	VAR robtarget Openhole_3455 := [[362.32, -32.55, 173.58], [-0.183051, 0.683002, 0.683002, 0.183051], [0,0,0,0], [9E9, 9E9, 9E9, 9E9, 9E9, 9E9]];
	VAR robtarget Openhole_3456 := [[362.32, -31.54, 174.16], [-0.183051, 0.683002, 0.683002, 0.183051], [0,0,0,0], [9E9, 9E9, 9E9, 9E9, 9E9, 9E9]];
	VAR robtarget Openhole_3457 := [[374.32, -31.54, 174.12], [-0.183051, 0.683002, 0.683002, 0.183051], [0,0,0,0], [9E9, 9E9, 9E9, 9E9, 9E9, 9E9]];
	VAR robtarget Openhole_3458 := [[389.32, -31.54, 174.07], [-0.146559, 0.691752, 0.6724, 0.218811], [0,0,0,0], [9E9, 9E9, 9E9, 9E9, 9E9, 9E9]];
	VAR robtarget Openhole_3459 := [[394.33, -31.54, 174.68], [-0.132991, 0.694488, 0.676088, 0.207135], [0,0,0,0], [9E9, 9E9, 9E9, 9E9, 9E9, 9E9]];
	VAR robtarget Openhole_3460 := [[394.83, -31.57, 174.72], [-0.131528, 0.694766, 0.676427, 0.206027], [0,0,0,0], [9E9, 9E9, 9E9, 9E9, 9E9, 9E9]];
	VAR robtarget Openhole_3461 := [[399.78, -32.12, 175.06], [-0.11586, 0.69755, 0.67957, 0.19541], [0,0,0,0], [9E9, 9E9, 9E9, 9E9, 9E9, 9E9]];
	VAR robtarget Openhole_3462 := [[407.69, -33.18, 175.63], [-0.089063, 0.701475, 0.684337, 0.177998], [0,0,0,0], [9E9, 9E9, 9E9, 9E9, 9E9, 9E9]];
	VAR robtarget Openhole_3463 := [[414.62, -33.85, 176.35], [-0.065291, 0.704086, 0.688563, 0.160875], [0,0,0,0], [9E9, 9E9, 9E9, 9E9, 9E9, 9E9]];
	VAR robtarget Openhole_3464 := [[420.07, -34.09, 177.06], [-0.04691, 0.705549, 0.691908, 0.145819], [0,0,0,0], [9E9, 9E9, 9E9, 9E9, 9E9, 9E9]];
	VAR robtarget Openhole_3465 := [[421.06, -34.1, 177.2], [-0.043641, 0.705759, 0.692517, 0.142901], [0,0,0,0], [9E9, 9E9, 9E9, 9E9, 9E9, 9E9]];
	VAR robtarget Openhole_3466 := [[421.55, -34.1, 177.27], [-0.042014, 0.705857, 0.69282, 0.141422], [0,0,0,0], [9E9, 9E9, 9E9, 9E9, 9E9, 9E9]];
	VAR robtarget Openhole_3467 := [[426.98, -33.88, 178.11], [-0.024649, 0.706677, 0.696114, 0.124201], [0,0,0,0], [9E9, 9E9, 9E9, 9E9, 9E9, 9E9]];
	VAR robtarget Openhole_3468 := [[436.34, -33.07, 179.54], [0.004362, 0.707093, 0.701125, 0.091781], [0,0,0,0], [9E9, 9E9, 9E9, 9E9, 9E9, 9E9]];
	VAR robtarget Openhole_3469 := [[438.32, -33.02, 179.82], [0.010929, 0.707022, 0.701966, 0.085107], [0,0,0,0], [9E9, 9E9, 9E9, 9E9, 9E9, 9E9]];
	VAR robtarget Openhole_3470 := [[438.81, -33.02, 179.88], [0.012627, 0.706994, 0.702162, 0.083481], [0,0,0,0], [9E9, 9E9, 9E9, 9E9, 9E9, 9E9]];
	VAR robtarget Openhole_3471 := [[439.31, -33.03, 179.95], [0.014351, 0.706961, 0.70235, 0.081878], [0,0,0,0], [9E9, 9E9, 9E9, 9E9, 9E9, 9E9]];
	VAR robtarget Openhole_3472 := [[442.77, -33.27, 180.4], [0.026976, 0.706592, 0.703516, 0.071171], [0,0,0,0], [9E9, 9E9, 9E9, 9E9, 9E9, 9E9]];
	VAR robtarget Openhole_3473 := [[447.66, -34.06, 181.06], [0.046306, 0.705589, 0.704776, 0.05736], [0,0,0,0], [9E9, 9E9, 9E9, 9E9, 9E9, 9E9]];
	VAR robtarget Openhole_3474 := [[448.16, -34.12, 181.13], [0.048183, 0.705463, 0.704893, 0.055904], [0,0,0,0], [9E9, 9E9, 9E9, 9E9, 9E9, 9E9]];
	VAR robtarget Openhole_3475 := [[448.65, -34.17, 181.2], [0.050018, 0.705336, 0.705011, 0.054399], [0,0,0,0], [9E9, 9E9, 9E9, 9E9, 9E9, 9E9]];
	VAR robtarget Openhole_3476 := [[449.14, -34.2, 181.27], [0.051809, 0.705206, 0.70513, 0.052839], [0,0,0,0], [9E9, 9E9, 9E9, 9E9, 9E9, 9E9]];
	VAR robtarget Openhole_3477 := [[449.64, -34.22, 181.34], [0.053533, 0.705077, 0.70525, 0.051209], [0,0,0,0], [9E9, 9E9, 9E9, 9E9, 9E9, 9E9]];
	VAR robtarget Openhole_3478 := [[450.13, -34.22, 181.42], [0.055212, 0.704948, 0.70537, 0.049531], [0,0,0,0], [9E9, 9E9, 9E9, 9E9, 9E9, 9E9]];
	VAR robtarget Openhole_3479 := [[450.63, -34.2, 181.49], [0.056822, 0.70482, 0.70549, 0.047788], [0,0,0,0], [9E9, 9E9, 9E9, 9E9, 9E9, 9E9]];
	VAR robtarget Openhole_3480 := [[451.12, -34.17, 181.56], [0.058384, 0.704692, 0.705609, 0.046], [0,0,0,0], [9E9, 9E9, 9E9, 9E9, 9E9, 9E9]];
	VAR robtarget Openhole_3481 := [[451.61, -34.11, 181.63], [0.05987, 0.704568, 0.705727, 0.04415], [0,0,0,0], [9E9, 9E9, 9E9, 9E9, 9E9, 9E9]];
	VAR robtarget Openhole_3482 := [[452.1, -34.05, 181.7], [0.061305, 0.704444, 0.705843, 0.042256], [0,0,0,0], [9E9, 9E9, 9E9, 9E9, 9E9, 9E9]];
	VAR robtarget Openhole_3483 := [[452.59, -33.96, 181.77], [0.062679, 0.704323, 0.705956, 0.040321], [0,0,0,0], [9E9, 9E9, 9E9, 9E9, 9E9, 9E9]];
	VAR robtarget Openhole_3484 := [[460.82, -32.06, 182.74], [0.083784, 0.702126, 0.707082, 0.005917], [0,0,0,0], [9E9, 9E9, 9E9, 9E9, 9E9, 9E9]];
	VAR robtarget Openhole_3485 := [[467.69, -30.95, 183.41], [0.102455, 0.699645, 0.706793, -0.021077], [0,0,0,0], [9E9, 9E9, 9E9, 9E9, 9E9, 9E9]];
	VAR robtarget Openhole_3486 := [[476.61, -29.98, 184.18], [0.127132, 0.695584, 0.705054, -0.053839], [0,0,0,0], [9E9, 9E9, 9E9, 9E9, 9E9, 9E9]];
	VAR robtarget Openhole_3487 := [[487.55, -29.21, 185.05], [0.156769, 0.68951, 0.701222, -0.091037], [0,0,0,0], [9E9, 9E9, 9E9, 9E9, 9E9, 9E9]];
	VAR robtarget Openhole_3488 := [[504.36, -28.38, 186.26], [0.198471, 0.678682, 0.692621, -0.142396], [0,0,0,0], [9E9, 9E9, 9E9, 9E9, 9E9, 9E9]];
	VAR robtarget Openhole_3489 := [[509.36, -28.38, 186.71], [0.183051, 0.683002, 0.683002, -0.183051], [0,0,0,0], [9E9, 9E9, 9E9, 9E9, 9E9, 9E9]];
	VAR robtarget Openhole_3490 := [[536.36, -28.38, 186.62], [0.183051, 0.683002, 0.683002, -0.183051], [0,0,0,0], [9E9, 9E9, 9E9, 9E9, 9E9, 9E9]];
	VAR robtarget Openhole_3491 := [[536.36, -27.26, 185.97], [0.183051, 0.683002, 0.683002, -0.183051], [0,0,0,0], [9E9, 9E9, 9E9, 9E9, 9E9, 9E9]];
	VAR robtarget Openhole_3492 := [[509.36, -27.26, 186.06], [0.183051, 0.683002, 0.683002, -0.183051], [0,0,0,0], [9E9, 9E9, 9E9, 9E9, 9E9, 9E9]];
	VAR robtarget Openhole_3493 := [[504.36, -27.26, 185.66], [0.195255, 0.679614, 0.691939, -0.14567], [0,0,0,0], [9E9, 9E9, 9E9, 9E9, 9E9, 9E9]];
	VAR robtarget Openhole_3494 := [[490.44, -27.87, 184.8], [0.160731, 0.688597, 0.699415, -0.104016], [0,0,0,0], [9E9, 9E9, 9E9, 9E9, 9E9, 9E9]];
	VAR robtarget Openhole_3495 := [[476.49, -28.59, 183.8], [0.122302, 0.69645, 0.704725, -0.057993], [0,0,0,0], [9E9, 9E9, 9E9, 9E9, 9E9, 9E9]];
	VAR robtarget Openhole_3496 := [[464.07, -29.6, 182.8], [0.086303, 0.70182, 0.706981, -0.013352], [0,0,0,0], [9E9, 9E9, 9E9, 9E9, 9E9, 9E9]];
	VAR robtarget Openhole_3497 := [[458.64, -30.3, 182.31], [0.070753, 0.703558, 0.707067, 0.007457], [0,0,0,0], [9E9, 9E9, 9E9, 9E9, 9E9, 9E9]];
	VAR robtarget Openhole_3498 := [[453.73, -31.11, 181.81], [0.057022, 0.704804, 0.706595, 0.026907], [0,0,0,0], [9E9, 9E9, 9E9, 9E9, 9E9, 9E9]];
	VAR robtarget Openhole_3499 := [[452.75, -31.23, 181.7], [0.054101, 0.705034, 0.706441, 0.030675], [0,0,0,0], [9E9, 9E9, 9E9, 9E9, 9E9, 9E9]];
	VAR robtarget Openhole_3500 := [[451.76, -31.32, 181.59], [0.051039, 0.705262, 0.706273, 0.034329], [0,0,0,0], [9E9, 9E9, 9E9, 9E9, 9E9, 9E9]];
	VAR robtarget Openhole_3501 := [[450.76, -31.35, 181.47], [0.0478, 0.705489, 0.706094, 0.037827], [0,0,0,0], [9E9, 9E9, 9E9, 9E9, 9E9, 9E9]];
	VAR robtarget Openhole_3502 := [[450.27, -31.35, 181.41], [0.046116, 0.705601, 0.706002, 0.039513], [0,0,0,0], [9E9, 9E9, 9E9, 9E9, 9E9, 9E9]];
	VAR robtarget Openhole_3503 := [[449.77, -31.34, 181.35], [0.044384, 0.705712, 0.705908, 0.041153], [0,0,0,0], [9E9, 9E9, 9E9, 9E9, 9E9, 9E9]];
	VAR robtarget Openhole_3504 := [[449.27, -31.31, 181.29], [0.042623, 0.705821, 0.705813, 0.042761], [0,0,0,0], [9E9, 9E9, 9E9, 9E9, 9E9, 9E9]];
	VAR robtarget Openhole_3505 := [[445.32, -30.96, 180.84], [0.02795, 0.706554, 0.704968, 0.054953], [0,0,0,0], [9E9, 9E9, 9E9, 9E9, 9E9, 9E9]];
	VAR robtarget Openhole_3506 := [[441.35, -30.75, 180.4], [0.01369, 0.706974, 0.703873, 0.067552], [0,0,0,0], [9E9, 9E9, 9E9, 9E9, 9E9, 9E9]];
	VAR robtarget Openhole_3507 := [[440.85, -30.75, 180.34], [0.011992, 0.707005, 0.703712, 0.069206], [0,0,0,0], [9E9, 9E9, 9E9, 9E9, 9E9, 9E9]];
	VAR robtarget Openhole_3508 := [[440.35, -30.75, 180.29], [0.010316, 0.707032, 0.703546, 0.070877], [0,0,0,0], [9E9, 9E9, 9E9, 9E9, 9E9, 9E9]];
	VAR robtarget Openhole_3509 := [[439.36, -30.78, 180.17], [0.007029, 0.707072, 0.703195, 0.074272], [0,0,0,0], [9E9, 9E9, 9E9, 9E9, 9E9, 9E9]];
	VAR robtarget Openhole_3510 := [[438.37, -30.84, 180.05], [0.003839, 0.707096, 0.702821, 0.077739], [0,0,0,0], [9E9, 9E9, 9E9, 9E9, 9E9, 9E9]];
	VAR robtarget Openhole_3511 := [[432.46, -31.52, 179.27], [-0.013978, 0.706969, 0.700109, 0.099234], [0,0,0,0], [9E9, 9E9, 9E9, 9E9, 9E9, 9E9]];
	VAR robtarget Openhole_3512 := [[426.07, -32.27, 178.34], [-0.032943, 0.706339, 0.696528, 0.121857], [0,0,0,0], [9E9, 9E9, 9E9, 9E9, 9E9, 9E9]];
	VAR robtarget Openhole_3513 := [[421.13, -32.53, 177.64], [-0.048461, 0.705444, 0.693564, 0.137728], [0,0,0,0], [9E9, 9E9, 9E9, 9E9, 9E9, 9E9]];
	VAR robtarget Openhole_3514 := [[419.64, -32.54, 177.44], [-0.05328, 0.705097, 0.692661, 0.142198], [0,0,0,0], [9E9, 9E9, 9E9, 9E9, 9E9, 9E9]];
	VAR robtarget Openhole_3515 := [[419.15, -32.54, 177.38], [-0.0549, 0.704972, 0.69236, 0.143659], [0,0,0,0], [9E9, 9E9, 9E9, 9E9, 9E9, 9E9]];
	VAR robtarget Openhole_3516 := [[413.19, -32.29, 176.69], [-0.074754, 0.703144, 0.688744, 0.1601], [0,0,0,0], [9E9, 9E9, 9E9, 9E9, 9E9, 9E9]];
	VAR robtarget Openhole_3517 := [[404.76, -31.51, 175.95], [-0.103082, 0.699553, 0.683609, 0.180772], [0,0,0,0], [9E9, 9E9, 9E9, 9E9, 9E9, 9E9]];
	VAR robtarget Openhole_3518 := [[397.32, -30.78, 175.42], [-0.126904, 0.695626, 0.678917, 0.197666], [0,0,0,0], [9E9, 9E9, 9E9, 9E9, 9E9, 9E9]];
	VAR robtarget Openhole_3519 := [[394.83, -30.66, 175.2], [-0.134181, 0.694259, 0.677213, 0.203426], [0,0,0,0], [9E9, 9E9, 9E9, 9E9, 9E9, 9E9]];
	VAR robtarget Openhole_3520 := [[389.32, -30.66, 174.58], [-0.149079, 0.691213, 0.673193, 0.216357], [0,0,0,0], [9E9, 9E9, 9E9, 9E9, 9E9, 9E9]];
	VAR robtarget Openhole_3521 := [[362.32, -30.66, 174.67], [-0.183051, 0.683002, 0.683002, 0.183051], [0,0,0,0], [9E9, 9E9, 9E9, 9E9, 9E9, 9E9]];
	VAR robtarget Openhole_3522 := [[362.33, -28.99, 175.63], [-0.183051, 0.683002, 0.683002, 0.183051], [0,0,0,0], [9E9, 9E9, 9E9, 9E9, 9E9, 9E9]];
	VAR robtarget Openhole_3523 := [[374.33, -28.99, 175.59], [-0.183051, 0.683002, 0.683002, 0.183051], [0,0,0,0], [9E9, 9E9, 9E9, 9E9, 9E9, 9E9]];
	VAR robtarget Openhole_3524 := [[389.33, -28.99, 175.55], [-0.153845, 0.690168, 0.674671, 0.211706], [0,0,0,0], [9E9, 9E9, 9E9, 9E9, 9E9, 9E9]];
	VAR robtarget Openhole_3525 := [[394.3, -28.99, 176.02], [-0.140535, 0.693001, 0.678257, 0.199918], [0,0,0,0], [9E9, 9E9, 9E9, 9E9, 9E9, 9E9]];
	VAR robtarget Openhole_3526 := [[394.82, -28.97, 176.09], [-0.139179, 0.693274, 0.67865, 0.198582], [0,0,0,0], [9E9, 9E9, 9E9, 9E9, 9E9, 9E9]];
	VAR robtarget Openhole_3527 := [[396.81, -28.94, 176.29], [-0.133756, 0.694341, 0.680085, 0.193609], [0,0,0,0], [9E9, 9E9, 9E9, 9E9, 9E9, 9E9]];
	VAR robtarget Openhole_3528 := [[397.31, -28.94, 176.34], [-0.132364, 0.694608, 0.680436, 0.19237], [0,0,0,0], [9E9, 9E9, 9E9, 9E9, 9E9, 9E9]];
	VAR robtarget Openhole_3529 := [[403.29, -29.19, 176.8], [-0.114504, 0.697774, 0.684397, 0.177765], [0,0,0,0], [9E9, 9E9, 9E9, 9E9, 9E9, 9E9]];
	VAR robtarget Openhole_3530 := [[414.23, -29.87, 177.64], [-0.079127, 0.702666, 0.691092, 0.149638], [0,0,0,0], [9E9, 9E9, 9E9, 9E9, 9E9, 9E9]];
	VAR robtarget Openhole_3531 := [[417.72, -29.94, 177.98], [-0.067846, 0.703844, 0.693168, 0.13971], [0,0,0,0], [9E9, 9E9, 9E9, 9E9, 9E9, 9E9]];
	VAR robtarget Openhole_3532 := [[418.21, -29.94, 178.03], [-0.06626, 0.703995, 0.693464, 0.138231], [0,0,0,0], [9E9, 9E9, 9E9, 9E9, 9E9, 9E9]];
	VAR robtarget Openhole_3533 := [[423.18, -29.75, 178.6], [-0.050752, 0.705283, 0.696384, 0.122678], [0,0,0,0], [9E9, 9E9, 9E9, 9E9, 9E9, 9E9]];
	VAR robtarget Openhole_3534 := [[427.61, -29.25, 179.16], [-0.037763, 0.706098, 0.698926, 0.107249], [0,0,0,0], [9E9, 9E9, 9E9, 9E9, 9E9, 9E9]];
	VAR robtarget Openhole_3535 := [[431.99, -28.38, 179.74], [-0.025976, 0.70663, 0.701298, 0.09045], [0,0,0,0], [9E9, 9E9, 9E9, 9E9, 9E9, 9E9]];
	VAR robtarget Openhole_3536 := [[436.77, -27.04, 180.33], [-0.014315, 0.706962, 0.703594, 0.070396], [0,0,0,0], [9E9, 9E9, 9E9, 9E9, 9E9, 9E9]];
	VAR robtarget Openhole_3537 := [[439.61, -26.14, 180.64], [-0.0077, 0.707065, 0.70473, 0.057931], [0,0,0,0], [9E9, 9E9, 9E9, 9E9, 9E9, 9E9]];
	VAR robtarget Openhole_3538 := [[441.02, -25.65, 180.77], [-0.004587, 0.707092, 0.705225, 0.05155], [0,0,0,0], [9E9, 9E9, 9E9, 9E9, 9E9, 9E9]];
	VAR robtarget Openhole_3539 := [[441.49, -25.47, 180.81], [-0.003609, 0.707098, 0.70538, 0.04939], [0,0,0,0], [9E9, 9E9, 9E9, 9E9, 9E9, 9E9]];
	VAR robtarget Openhole_3540 := [[441.94, -25.27, 180.86], [-0.002738, 0.707101, 0.705531, 0.047182], [0,0,0,0], [9E9, 9E9, 9E9, 9E9, 9E9, 9E9]];
	VAR robtarget Openhole_3541 := [[442.83, -24.81, 180.94], [-0.00127, 0.707106, 0.705819, 0.04266], [0,0,0,0], [9E9, 9E9, 9E9, 9E9, 9E9, 9E9]];
	VAR robtarget Openhole_3542 := [[443.59, -24.26, 181.01], [-0.000556, 0.707107, 0.706072, 0.038232], [0,0,0,0], [9E9, 9E9, 9E9, 9E9, 9E9, 9E9]];
	VAR robtarget Openhole_3543 := [[445.39, -24.26, 181.1], [0.005592, 0.707085, 0.706376, 0.032131], [0,0,0,0], [9E9, 9E9, 9E9, 9E9, 9E9, 9E9]];
	VAR robtarget Openhole_3544 := [[443.96, -22.2, 181.14], [-0.006277, 0.707079, 0.706469, 0.030031], [0,0,0,0], [9E9, 9E9, 9E9, 9E9, 9E9, 9E9]];
	VAR robtarget Openhole_3545 := [[442.15, -22.2, 181.08], [-0.012413, 0.706998, 0.706183, 0.036126], [0,0,0,0], [9E9, 9E9, 9E9, 9E9, 9E9, 9E9]];
	VAR robtarget Openhole_3546 := [[441.31, -22.66, 181.02], [-0.013707, 0.706974, 0.705945, 0.040513], [0,0,0,0], [9E9, 9E9, 9E9, 9E9, 9E9, 9E9]];
	VAR robtarget Openhole_3547 := [[440.05, -23.46, 180.9], [-0.01527, 0.706942, 0.705512, 0.04746], [0,0,0,0], [9E9, 9E9, 9E9, 9E9, 9E9, 9E9]];
	VAR robtarget Openhole_3548 := [[439.62, -23.72, 180.86], [-0.015855, 0.706929, 0.705354, 0.049754], [0,0,0,0], [9E9, 9E9, 9E9, 9E9, 9E9, 9E9]];
	VAR robtarget Openhole_3549 := [[438.31, -24.43, 180.73], [-0.017925, 0.70688, 0.704844, 0.056527], [0,0,0,0], [9E9, 9E9, 9E9, 9E9, 9E9, 9E9]];
	VAR robtarget Openhole_3550 := [[435.13, -25.85, 180.37], [-0.023883, 0.706703, 0.703452, 0.071802], [0,0,0,0], [9E9, 9E9, 9E9, 9E9, 9E9, 9E9]];
	VAR robtarget Openhole_3551 := [[434.67, -26.03, 180.31], [-0.024835, 0.706671, 0.703232, 0.073926], [0,0,0,0], [9E9, 9E9, 9E9, 9E9, 9E9, 9E9]];
	VAR robtarget Openhole_3552 := [[433.73, -26.37, 180.2], [-0.026829, 0.706598, 0.702778, 0.078118], [0,0,0,0], [9E9, 9E9, 9E9, 9E9, 9E9, 9E9]];
	VAR robtarget Openhole_3553 := [[432.32, -26.83, 180.02], [-0.030072, 0.706467, 0.70207, 0.084249], [0,0,0,0], [9E9, 9E9, 9E9, 9E9, 9E9, 9E9]];
	VAR robtarget Openhole_3554 := [[430.4, -27.35, 179.78], [-0.03475, 0.706252, 0.701076, 0.092158], [0,0,0,0], [9E9, 9E9, 9E9, 9E9, 9E9, 9E9]];
	VAR robtarget Openhole_3555 := [[427, -28.06, 179.36], [-0.043712, 0.705754, 0.699221, 0.105306], [0,0,0,0], [9E9, 9E9, 9E9, 9E9, 9E9, 9E9]];
	VAR robtarget Openhole_3556 := [[422.56, -28.57, 178.84], [-0.056642, 0.704835, 0.69672, 0.120752], [0,0,0,0], [9E9, 9E9, 9E9, 9E9, 9E9, 9E9]];
	VAR robtarget Openhole_3557 := [[417.09, -28.75, 178.28], [-0.073676, 0.703258, 0.693553, 0.137783], [0,0,0,0], [9E9, 9E9, 9E9, 9E9, 9E9, 9E9]];
	VAR robtarget Openhole_3558 := [[416.59, -28.75, 178.24], [-0.07526, 0.70309, 0.693261, 0.139247], [0,0,0,0], [9E9, 9E9, 9E9, 9E9, 9E9, 9E9]];
	VAR robtarget Openhole_3559 := [[408.63, -28.45, 177.61], [-0.100918, 0.699868, 0.688515, 0.161083], [0,0,0,0], [9E9, 9E9, 9E9, 9E9, 9E9, 9E9]];
	VAR robtarget Openhole_3560 := [[399.66, -28.03, 177], [-0.128482, 0.695336, 0.682809, 0.183772], [0,0,0,0], [9E9, 9E9, 9E9, 9E9, 9E9, 9E9]];
	VAR robtarget Openhole_3561 := [[398.16, -28.02, 176.87], [-0.132736, 0.694537, 0.681783, 0.187543], [0,0,0,0], [9E9, 9E9, 9E9, 9E9, 9E9, 9E9]];
	VAR robtarget Openhole_3562 := [[397.66, -28.02, 176.83], [-0.134118, 0.694271, 0.681433, 0.188811], [0,0,0,0], [9E9, 9E9, 9E9, 9E9, 9E9, 9E9]];
	VAR robtarget Openhole_3563 := [[395.18, -28.08, 176.58], [-0.140809, 0.692945, 0.679635, 0.195184], [0,0,0,0], [9E9, 9E9, 9E9, 9E9, 9E9, 9E9]];
	VAR robtarget Openhole_3564 := [[394.33, -28.09, 176.5], [-0.143106, 0.692474, 0.679032, 0.197269], [0,0,0,0], [9E9, 9E9, 9E9, 9E9, 9E9, 9E9]];
	VAR robtarget Openhole_3565 := [[389.33, -28.09, 176.07], [-0.156423, 0.689588, 0.675457, 0.209183], [0,0,0,0], [9E9, 9E9, 9E9, 9E9, 9E9, 9E9]];
	VAR robtarget Openhole_3566 := [[362.33, -28.09, 176.15], [-0.183051, 0.683002, 0.683002, 0.183051], [0,0,0,0], [9E9, 9E9, 9E9, 9E9, 9E9, 9E9]];
	VAR robtarget Openhole_3567 := [[362.33, -27.21, 176.66], [-0.183051, 0.683002, 0.683002, 0.183051], [0,0,0,0], [9E9, 9E9, 9E9, 9E9, 9E9, 9E9]];
	VAR robtarget Openhole_3568 := [[374.33, -27.21, 176.62], [-0.183051, 0.683002, 0.683002, 0.183051], [0,0,0,0], [9E9, 9E9, 9E9, 9E9, 9E9, 9E9]];
	VAR robtarget Openhole_3569 := [[389.33, -27.21, 176.58], [-0.158946, 0.689011, 0.676219, 0.206709], [0,0,0,0], [9E9, 9E9, 9E9, 9E9, 9E9, 9E9]];
	VAR robtarget Openhole_3570 := [[394.26, -27.21, 176.97], [-0.1459, 0.691891, 0.679711, 0.194917], [0,0,0,0], [9E9, 9E9, 9E9, 9E9, 9E9, 9E9]];
	VAR robtarget Openhole_3571 := [[399.8, -27.04, 177.48], [-0.13105, 0.694857, 0.683691, 0.180463], [0,0,0,0], [9E9, 9E9, 9E9, 9E9, 9E9, 9E9]];
	VAR robtarget Openhole_3572 := [[400.3, -27.04, 177.52], [-0.129638, 0.695122, 0.68403, 0.179173], [0,0,0,0], [9E9, 9E9, 9E9, 9E9, 9E9, 9E9]];
	VAR robtarget Openhole_3573 := [[416.26, -27.54, 178.59], [-0.080198, 0.702544, 0.693822, 0.136421], [0,0,0,0], [9E9, 9E9, 9E9, 9E9, 9E9, 9E9]];
	VAR robtarget Openhole_3574 := [[416.76, -27.54, 178.63], [-0.078618, 0.702723, 0.694109, 0.134954], [0,0,0,0], [9E9, 9E9, 9E9, 9E9, 9E9, 9E9]];
	VAR robtarget Openhole_3575 := [[417.26, -27.54, 178.67], [-0.077046, 0.702897, 0.694396, 0.133471], [0,0,0,0], [9E9, 9E9, 9E9, 9E9, 9E9, 9E9]];
	VAR robtarget Openhole_3576 := [[422.73, -27.32, 179.18], [-0.060159, 0.704543, 0.697489, 0.116231], [0,0,0,0], [9E9, 9E9, 9E9, 9E9, 9E9, 9E9]];
	VAR robtarget Openhole_3577 := [[426.68, -26.85, 179.6], [-0.048784, 0.705422, 0.699657, 0.102374], [0,0,0,0], [9E9, 9E9, 9E9, 9E9, 9E9, 9E9]];
	VAR robtarget Openhole_3578 := [[430.07, -26.09, 179.99], [-0.040036, 0.705972, 0.701473, 0.08908], [0,0,0,0], [9E9, 9E9, 9E9, 9E9, 9E9, 9E9]];
	VAR robtarget Openhole_3579 := [[432.91, -25.19, 180.33], [-0.033566, 0.70631, 0.702915, 0.07688], [0,0,0,0], [9E9, 9E9, 9E9, 9E9, 9E9, 9E9]];
	VAR robtarget Openhole_3580 := [[433.37, -25.01, 180.38], [-0.03261, 0.706354, 0.703143, 0.07477], [0,0,0,0], [9E9, 9E9, 9E9, 9E9, 9E9, 9E9]];
	VAR robtarget Openhole_3581 := [[433.83, -24.82, 180.44], [-0.0317, 0.706396, 0.703366, 0.072635], [0,0,0,0], [9E9, 9E9, 9E9, 9E9, 9E9, 9E9]];
	VAR robtarget Openhole_3582 := [[434.29, -24.62, 180.49], [-0.03083, 0.706434, 0.703586, 0.070479], [0,0,0,0], [9E9, 9E9, 9E9, 9E9, 9E9, 9E9]];
	VAR robtarget Openhole_3583 := [[435.19, -24.2, 180.6], [-0.029206, 0.706503, 0.70401, 0.06611], [0,0,0,0], [9E9, 9E9, 9E9, 9E9, 9E9, 9E9]];
	VAR robtarget Openhole_3584 := [[436.52, -23.52, 180.75], [-0.027018, 0.70659, 0.704604, 0.059438], [0,0,0,0], [9E9, 9E9, 9E9, 9E9, 9E9, 9E9]];
	VAR robtarget Openhole_3585 := [[438.24, -22.52, 180.93], [-0.024589, 0.706679, 0.705313, 0.050341], [0,0,0,0], [9E9, 9E9, 9E9, 9E9, 9E9, 9E9]];
	VAR robtarget Openhole_3586 := [[440.79, -20.96, 181.14], [-0.021236, 0.706788, 0.706163, 0.036515], [0,0,0,0], [9E9, 9E9, 9E9, 9E9, 9E9, 9E9]];
	VAR robtarget Openhole_3587 := [[441.58, -20.63, 181.18], [-0.01967, 0.706833, 0.706349, 0.032734], [0,0,0,0], [9E9, 9E9, 9E9, 9E9, 9E9, 9E9]];
	VAR robtarget Openhole_3588 := [[443.72, -20.63, 181.21], [-0.0124, 0.706998, 0.706647, 0.025499], [0,0,0,0], [9E9, 9E9, 9E9, 9E9, 9E9, 9E9]];
	VAR robtarget Openhole_3589 := [[443.53, -19.52, 181.27], [-0.016836, 0.706906, 0.706752, 0.022388], [0,0,0,0], [9E9, 9E9, 9E9, 9E9, 9E9, 9E9]];
	VAR robtarget Openhole_3590 := [[441.39, -19.52, 181.26], [-0.024098, 0.706696, 0.706486, 0.029628], [0,0,0,0], [9E9, 9E9, 9E9, 9E9, 9E9, 9E9]];
	VAR robtarget Openhole_3591 := [[440.77, -19.7, 181.25], [-0.025589, 0.706644, 0.706369, 0.032289], [0,0,0,0], [9E9, 9E9, 9E9, 9E9, 9E9, 9E9]];
	VAR robtarget Openhole_3592 := [[440.31, -19.89, 181.23], [-0.026469, 0.706611, 0.706264, 0.034505], [0,0,0,0], [9E9, 9E9, 9E9, 9E9, 9E9, 9E9]];
	VAR robtarget Openhole_3593 := [[439.86, -20.1, 181.2], [-0.027291, 0.70658, 0.706152, 0.03674], [0,0,0,0], [9E9, 9E9, 9E9, 9E9, 9E9, 9E9]];
	VAR robtarget Openhole_3594 := [[439.41, -20.32, 181.18], [-0.028065, 0.70655, 0.706031, 0.038988], [0,0,0,0], [9E9, 9E9, 9E9, 9E9, 9E9, 9E9]];
	VAR robtarget Openhole_3595 := [[438.97, -20.55, 181.15], [-0.028766, 0.706521, 0.705902, 0.041257], [0,0,0,0], [9E9, 9E9, 9E9, 9E9, 9E9, 9E9]];
	VAR robtarget Openhole_3596 := [[438.54, -20.81, 181.12], [-0.029338, 0.706498, 0.705764, 0.043559], [0,0,0,0], [9E9, 9E9, 9E9, 9E9, 9E9, 9E9]];
	VAR robtarget Openhole_3597 := [[436.45, -22.16, 180.91], [-0.031824, 0.70639, 0.704957, 0.055094], [0,0,0,0], [9E9, 9E9, 9E9, 9E9, 9E9, 9E9]];
	VAR robtarget Openhole_3598 := [[436.02, -22.42, 180.87], [-0.032422, 0.706363, 0.704776, 0.057366], [0,0,0,0], [9E9, 9E9, 9E9, 9E9, 9E9, 9E9]];
	VAR robtarget Openhole_3599 := [[435.15, -22.9, 180.77], [-0.033736, 0.706302, 0.704395, 0.061865], [0,0,0,0], [9E9, 9E9, 9E9, 9E9, 9E9, 9E9]];
	VAR robtarget Openhole_3600 := [[434.26, -23.35, 180.67], [-0.035204, 0.70623, 0.703992, 0.066298], [0,0,0,0], [9E9, 9E9, 9E9, 9E9, 9E9, 9E9]];
	VAR robtarget Openhole_3601 := [[433.36, -23.77, 180.57], [-0.036811, 0.706148, 0.703567, 0.070666], [0,0,0,0], [9E9, 9E9, 9E9, 9E9, 9E9, 9E9]];
	VAR robtarget Openhole_3602 := [[432.44, -24.15, 180.47], [-0.0386, 0.706052, 0.703124, 0.074945], [0,0,0,0], [9E9, 9E9, 9E9, 9E9, 9E9, 9E9]];
	VAR robtarget Openhole_3603 := [[431.98, -24.33, 180.42], [-0.039559, 0.705999, 0.702896, 0.077049], [0,0,0,0], [9E9, 9E9, 9E9, 9E9, 9E9, 9E9]];
	VAR robtarget Openhole_3604 := [[431.04, -24.65, 180.31], [-0.041636, 0.70588, 0.702433, 0.081169], [0,0,0,0], [9E9, 9E9, 9E9, 9E9, 9E9, 9E9]];
	VAR robtarget Openhole_3605 := [[428.64, -25.31, 180.05], [-0.047369, 0.705518, 0.701215, 0.091087], [0,0,0,0], [9E9, 9E9, 9E9, 9E9, 9E9, 9E9]];
	VAR robtarget Openhole_3606 := [[426.69, -25.72, 179.84], [-0.05246, 0.705158, 0.700197, 0.098614], [0,0,0,0], [9E9, 9E9, 9E9, 9E9, 9E9, 9E9]];
	VAR robtarget Openhole_3607 := [[422.74, -26.21, 179.46], [-0.063759, 0.704226, 0.698089, 0.11257], [0,0,0,0], [9E9, 9E9, 9E9, 9E9, 9E9, 9E9]];
	VAR robtarget Openhole_3608 := [[417.77, -26.42, 179.06], [-0.079038, 0.702676, 0.695353, 0.128391], [0,0,0,0], [9E9, 9E9, 9E9, 9E9, 9E9, 9E9]];
	VAR robtarget Openhole_3609 := [[416.77, -26.42, 178.98], [-0.082175, 0.702316, 0.694794, 0.13138], [0,0,0,0], [9E9, 9E9, 9E9, 9E9, 9E9, 9E9]];
	VAR robtarget Openhole_3610 := [[416.27, -26.42, 178.95], [-0.083749, 0.70213, 0.694514, 0.132856], [0,0,0,0], [9E9, 9E9, 9E9, 9E9, 9E9, 9E9]];
	VAR robtarget Openhole_3611 := [[401.3, -26.08, 178.04], [-0.129707, 0.695109, 0.685437, 0.173713], [0,0,0,0], [9E9, 9E9, 9E9, 9E9, 9E9, 9E9]];
	VAR robtarget Openhole_3612 := [[400.8, -26.08, 178.01], [-0.131118, 0.694844, 0.685102, 0.175029], [0,0,0,0], [9E9, 9E9, 9E9, 9E9, 9E9, 9E9]];
	VAR robtarget Openhole_3613 := [[395.33, -26.26, 177.54], [-0.14579, 0.691914, 0.681231, 0.189538], [0,0,0,0], [9E9, 9E9, 9E9, 9E9, 9E9, 9E9]];
	VAR robtarget Openhole_3614 := [[394.83, -26.28, 177.49], [-0.147053, 0.691647, 0.680863, 0.190853], [0,0,0,0], [9E9, 9E9, 9E9, 9E9, 9E9, 9E9]];
	VAR robtarget Openhole_3615 := [[394.33, -26.32, 177.44], [-0.148292, 0.691382, 0.680483, 0.192207], [0,0,0,0], [9E9, 9E9, 9E9, 9E9, 9E9, 9E9]];
	VAR robtarget Openhole_3616 := [[394.33, -26.32, 177.44], [-0.148274, 0.691386, 0.680487, 0.192192], [0,0,0,0], [9E9, 9E9, 9E9, 9E9, 9E9, 9E9]];
	VAR robtarget Openhole_3617 := [[389.33, -26.32, 177.09], [-0.161466, 0.688425, 0.67697, 0.204233], [0,0,0,0], [9E9, 9E9, 9E9, 9E9, 9E9, 9E9]];
	VAR robtarget Openhole_3618 := [[362.33, -26.32, 177.17], [-0.183051, 0.683002, 0.683002, 0.183051], [0,0,0,0], [9E9, 9E9, 9E9, 9E9, 9E9, 9E9]];
	VAR robtarget Openhole_3619 := [[362.34, -24.22, 178.39], [-0.183051, 0.683002, 0.683002, 0.183051], [0,0,0,0], [9E9, 9E9, 9E9, 9E9, 9E9, 9E9]];
	VAR robtarget Openhole_3620 := [[389.34, -24.22, 178.3], [-0.167484, 0.686986, 0.678732, 0.1983], [0,0,0,0], [9E9, 9E9, 9E9, 9E9, 9E9, 9E9]];
	VAR robtarget Openhole_3621 := [[394.34, -24.22, 178.55], [-0.154443, 0.690034, 0.682176, 0.186107], [0,0,0,0], [9E9, 9E9, 9E9, 9E9, 9E9, 9E9]];
	VAR robtarget Openhole_3622 := [[395.31, -24.2, 178.61], [-0.151914, 0.690595, 0.68285, 0.183618], [0,0,0,0], [9E9, 9E9, 9E9, 9E9, 9E9, 9E9]];
	VAR robtarget Openhole_3623 := [[401.29, -23.97, 179.01], [-0.136127, 0.69388, 0.68699, 0.167465], [0,0,0,0], [9E9, 9E9, 9E9, 9E9, 9E9, 9E9]];
	VAR robtarget Openhole_3624 := [[403.28, -23.96, 179.11], [-0.130503, 0.69496, 0.688285, 0.162062], [0,0,0,0], [9E9, 9E9, 9E9, 9E9, 9E9, 9E9]];
	VAR robtarget Openhole_3625 := [[403.78, -23.96, 179.14], [-0.129072, 0.695227, 0.688602, 0.160708], [0,0,0,0], [9E9, 9E9, 9E9, 9E9, 9E9, 9E9]];
	VAR robtarget Openhole_3626 := [[416.77, -24.13, 179.7], [-0.08952, 0.701417, 0.696131, 0.124106], [0,0,0,0], [9E9, 9E9, 9E9, 9E9, 9E9, 9E9]];
	VAR robtarget Openhole_3627 := [[417.27, -24.13, 179.73], [-0.087961, 0.701614, 0.696397, 0.122602], [0,0,0,0], [9E9, 9E9, 9E9, 9E9, 9E9, 9E9]];
	VAR robtarget Openhole_3628 := [[422.76, -23.95, 180.04], [-0.071101, 0.703523, 0.699235, 0.105216], [0,0,0,0], [9E9, 9E9, 9E9, 9E9, 9E9, 9E9]];
	VAR robtarget Openhole_3629 := [[426.72, -23.49, 180.33], [-0.059741, 0.704579, 0.701196, 0.091234], [0,0,0,0], [9E9, 9E9, 9E9, 9E9, 9E9, 9E9]];
	VAR robtarget Openhole_3630 := [[427.7, -23.31, 180.41], [-0.057123, 0.704796, 0.701671, 0.08751], [0,0,0,0], [9E9, 9E9, 9E9, 9E9, 9E9, 9E9]];
	VAR robtarget Openhole_3631 := [[428.19, -23.21, 180.45], [-0.055857, 0.704897, 0.701905, 0.085609], [0,0,0,0], [9E9, 9E9, 9E9, 9E9, 9E9, 9E9]];
	VAR robtarget Openhole_3632 := [[430.12, -22.73, 180.62], [-0.051069, 0.70526, 0.702816, 0.077781], [0,0,0,0], [9E9, 9E9, 9E9, 9E9, 9E9, 9E9]];
	VAR robtarget Openhole_3633 := [[430.6, -22.59, 180.66], [-0.049944, 0.705341, 0.703036, 0.075769], [0,0,0,0], [9E9, 9E9, 9E9, 9E9, 9E9, 9E9]];
	VAR robtarget Openhole_3634 := [[432.02, -22.13, 180.78], [-0.046757, 0.705559, 0.703673, 0.069601], [0,0,0,0], [9E9, 9E9, 9E9, 9E9, 9E9, 9E9]];
	VAR robtarget Openhole_3635 := [[432.49, -21.97, 180.82], [-0.045748, 0.705625, 0.703877, 0.067509], [0,0,0,0], [9E9, 9E9, 9E9, 9E9, 9E9, 9E9]];
	VAR robtarget Openhole_3636 := [[433.88, -21.41, 180.95], [-0.04298, 0.705799, 0.704463, 0.061087], [0,0,0,0], [9E9, 9E9, 9E9, 9E9, 9E9, 9E9]];
	VAR robtarget Openhole_3637 := [[434.78, -20.99, 181.03], [-0.041382, 0.705895, 0.704831, 0.056687], [0,0,0,0], [9E9, 9E9, 9E9, 9E9, 9E9, 9E9]];
	VAR robtarget Openhole_3638 := [[435.23, -20.76, 181.07], [-0.040664, 0.705937, 0.705007, 0.054452], [0,0,0,0], [9E9, 9E9, 9E9, 9E9, 9E9, 9E9]];
	VAR robtarget Openhole_3639 := [[436.1, -20.28, 181.14], [-0.039368, 0.70601, 0.705342, 0.049929], [0,0,0,0], [9E9, 9E9, 9E9, 9E9, 9E9, 9E9]];
	VAR robtarget Openhole_3640 := [[436.54, -20.05, 181.18], [-0.038673, 0.706048, 0.705498, 0.047676], [0,0,0,0], [9E9, 9E9, 9E9, 9E9, 9E9, 9E9]];
	VAR robtarget Openhole_3641 := [[436.99, -19.83, 181.21], [-0.037886, 0.706091, 0.705645, 0.045448], [0,0,0,0], [9E9, 9E9, 9E9, 9E9, 9E9, 9E9]];
	VAR robtarget Openhole_3642 := [[437.9, -19.41, 181.26], [-0.036244, 0.706177, 0.705917, 0.041007], [0,0,0,0], [9E9, 9E9, 9E9, 9E9, 9E9, 9E9]];
	VAR robtarget Openhole_3643 := [[438.36, -19.23, 181.28], [-0.035295, 0.706225, 0.70604, 0.038832], [0,0,0,0], [9E9, 9E9, 9E9, 9E9, 9E9, 9E9]];
	VAR robtarget Openhole_3644 := [[438.84, -19.07, 181.3], [-0.034249, 0.706277, 0.706154, 0.036699], [0,0,0,0], [9E9, 9E9, 9E9, 9E9, 9E9, 9E9]];
	VAR robtarget Openhole_3645 := [[439.31, -18.93, 181.31], [-0.033128, 0.70633, 0.70626, 0.034601], [0,0,0,0], [9E9, 9E9, 9E9, 9E9, 9E9, 9E9]];
	VAR robtarget Openhole_3646 := [[440.28, -18.68, 181.33], [-0.030699, 0.70644, 0.706449, 0.030501], [0,0,0,0], [9E9, 9E9, 9E9, 9E9, 9E9, 9E9]];
	VAR robtarget Openhole_3647 := [[440.77, -18.58, 181.34], [-0.029365, 0.706497, 0.706531, 0.028522], [0,0,0,0], [9E9, 9E9, 9E9, 9E9, 9E9, 9E9]];
	VAR robtarget Openhole_3648 := [[441.27, -18.53, 181.34], [-0.027847, 0.706558, 0.706603, 0.026677], [0,0,0,0], [9E9, 9E9, 9E9, 9E9, 9E9, 9E9]];
	VAR robtarget Openhole_3649 := [[441.35, -18.53, 181.34], [-0.027583, 0.706569, 0.706613, 0.026423], [0,0,0,0], [9E9, 9E9, 9E9, 9E9, 9E9, 9E9]];
	VAR robtarget Openhole_3650 := [[443.12, -18.53, 181.33], [-0.021572, 0.706778, 0.706812, 0.020421], [0,0,0,0], [9E9, 9E9, 9E9, 9E9, 9E9, 9E9]];
	VAR robtarget Openhole_3651 := [[443.2, -17.55, 181.39], [-0.024639, 0.706677, 0.706907, 0.016804], [0,0,0,0], [9E9, 9E9, 9E9, 9E9, 9E9, 9E9]];
	VAR robtarget Openhole_3652 := [[441.43, -17.55, 181.41], [-0.030646, 0.706442, 0.706739, 0.022811], [0,0,0,0], [9E9, 9E9, 9E9, 9E9, 9E9, 9E9]];
	VAR robtarget Openhole_3653 := [[441.37, -17.54, 181.42], [-0.030893, 0.706432, 0.706733, 0.022996], [0,0,0,0], [9E9, 9E9, 9E9, 9E9, 9E9, 9E9]];
	VAR robtarget Openhole_3654 := [[440.87, -17.63, 181.42], [-0.03227, 0.70637, 0.706667, 0.024948], [0,0,0,0], [9E9, 9E9, 9E9, 9E9, 9E9, 9E9]];
	VAR robtarget Openhole_3655 := [[436.92, -18.24, 181.4], [-0.043491, 0.705768, 0.705956, 0.04032], [0,0,0,0], [9E9, 9E9, 9E9, 9E9, 9E9, 9E9]];
	VAR robtarget Openhole_3656 := [[436.43, -18.34, 181.39], [-0.044804, 0.705686, 0.705841, 0.042288], [0,0,0,0], [9E9, 9E9, 9E9, 9E9, 9E9, 9E9]];
	VAR robtarget Openhole_3657 := [[435.94, -18.42, 181.38], [-0.046188, 0.705597, 0.705724, 0.044205], [0,0,0,0], [9E9, 9E9, 9E9, 9E9, 9E9, 9E9]];
	VAR robtarget Openhole_3658 := [[434.95, -18.6, 181.36], [-0.048855, 0.705417, 0.705469, 0.048095], [0,0,0,0], [9E9, 9E9, 9E9, 9E9, 9E9, 9E9]];
	VAR robtarget Openhole_3659 := [[434.46, -18.67, 181.35], [-0.050258, 0.705318, 0.705338, 0.049985], [0,0,0,0], [9E9, 9E9, 9E9, 9E9, 9E9, 9E9]];
	VAR robtarget Openhole_3660 := [[433.97, -18.76, 181.34], [-0.051617, 0.70522, 0.705199, 0.051901], [0,0,0,0], [9E9, 9E9, 9E9, 9E9, 9E9, 9E9]];
	VAR robtarget Openhole_3661 := [[430.5, -19.24, 181.26], [-0.061459, 0.704431, 0.704118, 0.064943], [0,0,0,0], [9E9, 9E9, 9E9, 9E9, 9E9, 9E9]];
	VAR robtarget Openhole_3662 := [[429.51, -19.35, 181.24], [-0.064344, 0.704173, 0.703775, 0.068564], [0,0,0,0], [9E9, 9E9, 9E9, 9E9, 9E9, 9E9]];
	VAR robtarget Openhole_3663 := [[429.01, -19.4, 181.23], [-0.065818, 0.704037, 0.7036, 0.07034], [0,0,0,0], [9E9, 9E9, 9E9, 9E9, 9E9, 9E9]];
	VAR robtarget Openhole_3664 := [[424.02, -19.61, 181.16], [-0.081306, 0.702417, 0.701724, 0.087084], [0,0,0,0], [9E9, 9E9, 9E9, 9E9, 9E9, 9E9]];
	VAR robtarget Openhole_3665 := [[422.52, -19.62, 181.15], [-0.086077, 0.701848, 0.701116, 0.091846], [0,0,0,0], [9E9, 9E9, 9E9, 9E9, 9E9, 9E9]];
	VAR robtarget Openhole_3666 := [[422.02, -19.61, 181.15], [-0.087674, 0.70165, 0.70091, 0.09341], [0,0,0,0], [9E9, 9E9, 9E9, 9E9, 9E9, 9E9]];
	VAR robtarget Openhole_3667 := [[407.52, -19.42, 181.14], [-0.132324, 0.694615, 0.693827, 0.136397], [0,0,0,0], [9E9, 9E9, 9E9, 9E9, 9E9, 9E9]];
	VAR robtarget Openhole_3668 := [[407.02, -19.42, 181.14], [-0.133765, 0.694339, 0.693545, 0.137826], [0,0,0,0], [9E9, 9E9, 9E9, 9E9, 9E9, 9E9]];
	VAR robtarget Openhole_3669 := [[398.02, -19.61, 181.01], [-0.158222, 0.689178, 0.688032, 0.163131], [0,0,0,0], [9E9, 9E9, 9E9, 9E9, 9E9, 9E9]];
	VAR robtarget Openhole_3670 := [[394.34, -19.81, 180.89], [-0.167354, 0.687017, 0.685546, 0.173283], [0,0,0,0], [9E9, 9E9, 9E9, 9E9, 9E9, 9E9]];
	VAR robtarget Openhole_3671 := [[362.34, -19.81, 180.93], [-0.183051, 0.683002, 0.683002, 0.183051], [0,0,0,0], [9E9, 9E9, 9E9, 9E9, 9E9, 9E9]];
	VAR robtarget Openhole_3672 := [[362.35, -16.66, 182.75], [-0.183051, 0.683002, 0.683002, 0.183051], [0,0,0,0], [9E9, 9E9, 9E9, 9E9, 9E9, 9E9]];
	VAR robtarget Openhole_3673 := [[389.35, -16.66, 182.67], [-0.189033, 0.681371, 0.684641, 0.176826], [0,0,0,0], [9E9, 9E9, 9E9, 9E9, 9E9, 9E9]];
	VAR robtarget Openhole_3674 := [[394.35, -16.66, 182.55], [-0.17654, 0.684714, 0.687805, 0.164087], [0,0,0,0], [9E9, 9E9, 9E9, 9E9, 9E9, 9E9]];
	VAR robtarget Openhole_3675 := [[395.16, -16.63, 182.55], [-0.174561, 0.685222, 0.688324, 0.161894], [0,0,0,0], [9E9, 9E9, 9E9, 9E9, 9E9, 9E9]];
	VAR robtarget Openhole_3676 := [[403.65, -16.31, 182.49], [-0.152823, 0.690395, 0.693542, 0.137838], [0,0,0,0], [9E9, 9E9, 9E9, 9E9, 9E9, 9E9]];
	VAR robtarget Openhole_3677 := [[410.15, -16.25, 182.35], [-0.134604, 0.694177, 0.697045, 0.118862], [0,0,0,0], [9E9, 9E9, 9E9, 9E9, 9E9, 9E9]];
	VAR robtarget Openhole_3678 := [[410.65, -16.25, 182.34], [-0.133147, 0.694458, 0.697296, 0.117383], [0,0,0,0], [9E9, 9E9, 9E9, 9E9, 9E9, 9E9]];
	VAR robtarget Openhole_3679 := [[425.64, -16.49, 181.88], [-0.086387, 0.70181, 0.703469, 0.071638], [0,0,0,0], [9E9, 9E9, 9E9, 9E9, 9E9, 9E9]];
	VAR robtarget Openhole_3680 := [[437.63, -16.79, 181.55], [-0.046017, 0.705608, 0.706334, 0.033055], [0,0,0,0], [9E9, 9E9, 9E9, 9E9, 9E9, 9E9]];
	VAR robtarget Openhole_3681 := [[438.13, -16.79, 181.54], [-0.04435, 0.705715, 0.706411, 0.031365], [0,0,0,0], [9E9, 9E9, 9E9, 9E9, 9E9, 9E9]];
	VAR robtarget Openhole_3682 := [[438.63, -16.79, 181.53], [-0.042674, 0.705818, 0.706484, 0.029681], [0,0,0,0], [9E9, 9E9, 9E9, 9E9, 9E9, 9E9]];
	VAR robtarget Openhole_3683 := [[440.13, -16.73, 181.51], [-0.037825, 0.706094, 0.706684, 0.024434], [0,0,0,0], [9E9, 9E9, 9E9, 9E9, 9E9, 9E9]];
	VAR robtarget Openhole_3684 := [[440.63, -16.69, 181.5], [-0.036278, 0.706176, 0.706745, 0.022617], [0,0,0,0], [9E9, 9E9, 9E9, 9E9, 9E9, 9E9]];
	VAR robtarget Openhole_3685 := [[441.11, -16.58, 181.5], [-0.035012, 0.706239, 0.706807, 0.020591], [0,0,0,0], [9E9, 9E9, 9E9, 9E9, 9E9, 9E9]];
	VAR robtarget Openhole_3686 := [[441.66, -16.48, 181.49], [-0.033486, 0.706313, 0.706867, 0.018418], [0,0,0,0], [9E9, 9E9, 9E9, 9E9, 9E9, 9E9]];
	VAR robtarget Openhole_3687 := [[443.56, -16.48, 181.44], [-0.027068, 0.706589, 0.707005, 0.011989], [0,0,0,0], [9E9, 9E9, 9E9, 9E9, 9E9, 9E9]];
	VAR robtarget Openhole_3688 := [[443.93, -15.46, 181.49], [-0.029287, 0.7065, 0.70707, 0.007235], [0,0,0,0], [9E9, 9E9, 9E9, 9E9, 9E9, 9E9]];
	VAR robtarget Openhole_3689 := [[442.03, -15.46, 181.55], [-0.035703, 0.706205, 0.706975, 0.01367], [0,0,0,0], [9E9, 9E9, 9E9, 9E9, 9E9, 9E9]];
	VAR robtarget Openhole_3690 := [[441.46, -15.51, 181.57], [-0.037458, 0.706114, 0.706931, 0.015782], [0,0,0,0], [9E9, 9E9, 9E9, 9E9, 9E9, 9E9]];
	VAR robtarget Openhole_3691 := [[440.97, -15.59, 181.58], [-0.038827, 0.70604, 0.706884, 0.017742], [0,0,0,0], [9E9, 9E9, 9E9, 9E9, 9E9, 9E9]];
	VAR robtarget Openhole_3692 := [[439.97, -15.62, 181.61], [-0.042093, 0.705853, 0.706788, 0.021221], [0,0,0,0], [9E9, 9E9, 9E9, 9E9, 9E9, 9E9]];
	VAR robtarget Openhole_3693 := [[439.47, -15.62, 181.63], [-0.043787, 0.70575, 0.706736, 0.022896], [0,0,0,0], [9E9, 9E9, 9E9, 9E9, 9E9, 9E9]];
	VAR robtarget Openhole_3694 := [[438.97, -15.61, 181.64], [-0.045514, 0.70564, 0.706681, 0.024532], [0,0,0,0], [9E9, 9E9, 9E9, 9E9, 9E9, 9E9]];
	VAR robtarget Openhole_3695 := [[438.47, -15.58, 181.66], [-0.047274, 0.705525, 0.706624, 0.02613], [0,0,0,0], [9E9, 9E9, 9E9, 9E9, 9E9, 9E9]];
	VAR robtarget Openhole_3696 := [[437.48, -15.49, 181.71], [-0.050897, 0.705273, 0.706504, 0.02919], [0,0,0,0], [9E9, 9E9, 9E9, 9E9, 9E9, 9E9]];
	VAR robtarget Openhole_3697 := [[431.51, -14.94, 182], [-0.072517, 0.703378, 0.705526, 0.047249], [0,0,0,0], [9E9, 9E9, 9E9, 9E9, 9E9, 9E9]];
	VAR robtarget Openhole_3698 := [[422.53, -14.66, 182.43], [-0.102246, 0.699676, 0.703052, 0.075619], [0,0,0,0], [9E9, 9E9, 9E9, 9E9, 9E9, 9E9]];
	VAR robtarget Openhole_3699 := [[413.54, -14.6, 182.83], [-0.129852, 0.695082, 0.699492, 0.103495], [0,0,0,0], [9E9, 9E9, 9E9, 9E9, 9E9, 9E9]];
	VAR robtarget Openhole_3700 := [[413.04, -14.6, 182.85], [-0.131325, 0.694805, 0.699265, 0.105014], [0,0,0,0], [9E9, 9E9, 9E9, 9E9, 9E9, 9E9]];
	VAR robtarget Openhole_3701 := [[401.55, -14.77, 183.26], [-0.163243, 0.688006, 0.693301, 0.139045], [0,0,0,0], [9E9, 9E9, 9E9, 9E9, 9E9, 9E9]];
	VAR robtarget Openhole_3702 := [[394.35, -15.07, 183.39], [-0.181155, 0.683508, 0.688896, 0.159443], [0,0,0,0], [9E9, 9E9, 9E9, 9E9, 9E9, 9E9]];
	VAR robtarget Openhole_3703 := [[389.35, -15.07, 183.58], [-0.193533, 0.680107, 0.685795, 0.172295], [0,0,0,0], [9E9, 9E9, 9E9, 9E9, 9E9, 9E9]];
	VAR robtarget Openhole_3704 := [[362.35, -15.07, 183.67], [-0.183051, 0.683002, 0.683002, 0.183051], [0,0,0,0], [9E9, 9E9, 9E9, 9E9, 9E9, 9E9]];
	VAR robtarget Openhole_3705 := [[362.35, -14.11, 184.23], [-0.183051, 0.683002, 0.683002, 0.183051], [0,0,0,0], [9E9, 9E9, 9E9, 9E9, 9E9, 9E9]];
	VAR robtarget Openhole_3706 := [[389.35, -14.11, 184.14], [-0.196264, 0.679324, 0.686481, 0.169539], [0,0,0,0], [9E9, 9E9, 9E9, 9E9, 9E9, 9E9]];
	VAR robtarget Openhole_3707 := [[394.35, -14.11, 183.9], [-0.183956, 0.682759, 0.689544, 0.156617], [0,0,0,0], [9E9, 9E9, 9E9, 9E9, 9E9, 9E9]];
	VAR robtarget Openhole_3708 := [[404.57, -13.71, 183.59], [-0.158197, 0.689183, 0.69556, 0.127266], [0,0,0,0], [9E9, 9E9, 9E9, 9E9, 9E9, 9E9]];
	VAR robtarget Openhole_3709 := [[419.55, -13.55, 182.87], [-0.115078, 0.69768, 0.702399, 0.081456], [0,0,0,0], [9E9, 9E9, 9E9, 9E9, 9E9, 9E9]];
	VAR robtarget Openhole_3710 := [[420.05, -13.55, 182.85], [-0.113543, 0.697931, 0.702581, 0.079876], [0,0,0,0], [9E9, 9E9, 9E9, 9E9, 9E9, 9E9]];
	VAR robtarget Openhole_3711 := [[430.53, -13.69, 182.27], [-0.079851, 0.702584, 0.705587, 0.046339], [0,0,0,0], [9E9, 9E9, 9E9, 9E9, 9E9, 9E9]];
	VAR robtarget Openhole_3712 := [[435.51, -14.05, 181.96], [-0.062314, 0.704356, 0.70643, 0.030925], [0,0,0,0], [9E9, 9E9, 9E9, 9E9, 9E9, 9E9]];
	VAR robtarget Openhole_3713 := [[438.48, -14.4, 181.78], [-0.051201, 0.705251, 0.706761, 0.022123], [0,0,0,0], [9E9, 9E9, 9E9, 9E9, 9E9, 9E9]];
	VAR robtarget Openhole_3714 := [[438.98, -14.45, 181.76], [-0.04939, 0.70538, 0.706807, 0.020588], [0,0,0,0], [9E9, 9E9, 9E9, 9E9, 9E9, 9E9]];
	VAR robtarget Openhole_3715 := [[439.48, -14.47, 181.73], [-0.047627, 0.705501, 0.706852, 0.018992], [0,0,0,0], [9E9, 9E9, 9E9, 9E9, 9E9, 9E9]];
	VAR robtarget Openhole_3716 := [[439.98, -14.49, 181.71], [-0.045913, 0.705615, 0.706894, 0.01734], [0,0,0,0], [9E9, 9E9, 9E9, 9E9, 9E9, 9E9]];
	VAR robtarget Openhole_3717 := [[440.98, -14.49, 181.67], [-0.042535, 0.705826, 0.706969, 0.013974], [0,0,0,0], [9E9, 9E9, 9E9, 9E9, 9E9, 9E9]];
	VAR robtarget Openhole_3718 := [[441.98, -14.53, 181.62], [-0.039029, 0.706029, 0.707025, 0.010732], [0,0,0,0], [9E9, 9E9, 9E9, 9E9, 9E9, 9E9]];
	VAR robtarget Openhole_3719 := [[442.51, -14.54, 181.6], [-0.037183, 0.706128, 0.70705, 0.008962], [0,0,0,0], [9E9, 9E9, 9E9, 9E9, 9E9, 9E9]];
	VAR robtarget Openhole_3720 := [[444.28, -14.54, 181.52], [-0.031181, 0.706419, 0.707101, 0.002936], [0,0,0,0], [9E9, 9E9, 9E9, 9E9, 9E9, 9E9]];
	VAR robtarget Openhole_3721 := [[445.21, -13.31, 181.53], [-0.032234, 0.706372, 0.707093, -0.004392], [0,0,0,0], [9E9, 9E9, 9E9, 9E9, 9E9, 9E9]];
	VAR robtarget Openhole_3722 := [[443.43, -13.31, 181.63], [-0.03824, 0.706072, 0.707105, 0.001641], [0,0,0,0], [9E9, 9E9, 9E9, 9E9, 9E9, 9E9]];
	VAR robtarget Openhole_3723 := [[442.74, -13.1, 181.68], [-0.041273, 0.705901, 0.707099, 0.003287], [0,0,0,0], [9E9, 9E9, 9E9, 9E9, 9E9, 9E9]];
	VAR robtarget Openhole_3724 := [[440.25, -13.05, 181.83], [-0.049868, 0.705346, 0.707012, 0.011561], [0,0,0,0], [9E9, 9E9, 9E9, 9E9, 9E9, 9E9]];
	VAR robtarget Openhole_3725 := [[433.78, -12.57, 182.27], [-0.072956, 0.703333, 0.706392, 0.031776], [0,0,0,0], [9E9, 9E9, 9E9, 9E9, 9E9, 9E9]];
	VAR robtarget Openhole_3726 := [[427.8, -12.45, 182.66], [-0.092777, 0.700994, 0.705246, 0.051262], [0,0,0,0], [9E9, 9E9, 9E9, 9E9, 9E9, 9E9]];
	VAR robtarget Openhole_3727 := [[427.3, -12.45, 182.7], [-0.094372, 0.700781, 0.705125, 0.052902], [0,0,0,0], [9E9, 9E9, 9E9, 9E9, 9E9, 9E9]];
	VAR robtarget Openhole_3728 := [[408.83, -12.69, 183.77], [-0.14945, 0.691133, 0.698238, 0.111639], [0,0,0,0], [9E9, 9E9, 9E9, 9E9, 9E9, 9E9]];
	VAR robtarget Openhole_3729 := [[397.35, -13.06, 184.29], [-0.17938, 0.683976, 0.691975, 0.145503], [0,0,0,0], [9E9, 9E9, 9E9, 9E9, 9E9, 9E9]];
	VAR robtarget Openhole_3730 := [[394.33, -13.23, 184.37], [-0.186569, 0.68205, 0.690114, 0.154087], [0,0,0,0], [9E9, 9E9, 9E9, 9E9, 9E9, 9E9]];
	VAR robtarget Openhole_3731 := [[389.36, -13.23, 184.65], [-0.198759, 0.678598, 0.6871, 0.167014], [0,0,0,0], [9E9, 9E9, 9E9, 9E9, 9E9, 9E9]];
	VAR robtarget Openhole_3732 := [[362.36, -13.23, 184.74], [-0.183051, 0.683002, 0.683002, 0.183051], [0,0,0,0], [9E9, 9E9, 9E9, 9E9, 9E9, 9E9]];
	VAR robtarget Openhole_3733 := [[362.36, -12.34, 185.25], [-0.183051, 0.683002, 0.683002, 0.183051], [0,0,0,0], [9E9, 9E9, 9E9, 9E9, 9E9, 9E9]];
	VAR robtarget Openhole_3734 := [[374.36, -12.34, 185.21], [-0.183051, 0.683002, 0.683002, 0.183051], [0,0,0,0], [9E9, 9E9, 9E9, 9E9, 9E9, 9E9]];
	VAR robtarget Openhole_3735 := [[389.36, -12.34, 185.16], [-0.201251, 0.677863, 0.687709, 0.164489], [0,0,0,0], [9E9, 9E9, 9E9, 9E9, 9E9, 9E9]];
	VAR robtarget Openhole_3736 := [[394.34, -12.34, 184.84], [-0.189119, 0.681347, 0.690688, 0.151493], [0,0,0,0], [9E9, 9E9, 9E9, 9E9, 9E9, 9E9]];
	VAR robtarget Openhole_3737 := [[404.84, -11.88, 184.36], [-0.163039, 0.688054, 0.696696, 0.120889], [0,0,0,0], [9E9, 9E9, 9E9, 9E9, 9E9, 9E9]];
	VAR robtarget Openhole_3738 := [[429.78, -11.27, 182.76], [-0.090335, 0.701313, 0.705929, 0.040793], [0,0,0,0], [9E9, 9E9, 9E9, 9E9, 9E9, 9E9]];
	VAR robtarget Openhole_3739 := [[431.77, -11.25, 182.62], [-0.083929, 0.702108, 0.706284, 0.034099], [0,0,0,0], [9E9, 9E9, 9E9, 9E9, 9E9, 9E9]];
	VAR robtarget Openhole_3740 := [[432.27, -11.25, 182.58], [-0.082304, 0.702301, 0.706363, 0.032434], [0,0,0,0], [9E9, 9E9, 9E9, 9E9, 9E9, 9E9]];
	VAR robtarget Openhole_3741 := [[441.74, -11.43, 181.86], [-0.050325, 0.705314, 0.707106, 0.00103], [0,0,0,0], [9E9, 9E9, 9E9, 9E9, 9E9, 9E9]];
	VAR robtarget Openhole_3742 := [[442.24, -11.45, 181.82], [-0.048561, 0.705437, 0.707107, -0.000574], [0,0,0,0], [9E9, 9E9, 9E9, 9E9, 9E9, 9E9]];
	VAR robtarget Openhole_3743 := [[443.23, -11.52, 181.74], [-0.044965, 0.705676, 0.707097, -0.003712], [0,0,0,0], [9E9, 9E9, 9E9, 9E9, 9E9, 9E9]];
	VAR robtarget Openhole_3744 := [[444.22, -11.62, 181.67], [-0.04128, 0.705901, 0.707075, -0.006756], [0,0,0,0], [9E9, 9E9, 9E9, 9E9, 9E9, 9E9]];
	VAR robtarget Openhole_3745 := [[444.72, -11.69, 181.63], [-0.039394, 0.706009, 0.707059, -0.008227], [0,0,0,0], [9E9, 9E9, 9E9, 9E9, 9E9, 9E9]];
	VAR robtarget Openhole_3746 := [[445.25, -11.83, 181.59], [-0.037109, 0.706132, 0.707042, -0.009568], [0,0,0,0], [9E9, 9E9, 9E9, 9E9, 9E9, 9E9]];
	VAR robtarget Openhole_3747 := [[454.82, -12.87, 180.98], [-0.001006, 0.707106, 0.706056, -0.038538], [0,0,0,0], [9E9, 9E9, 9E9, 9E9, 9E9, 9E9]];
	VAR robtarget Openhole_3748 := [[455.36, -12.53, 180.93], [-0.00035, 0.707107, 0.705889, -0.041479], [0,0,0,0], [9E9, 9E9, 9E9, 9E9, 9E9, 9E9]];
	VAR robtarget Openhole_3749 := [[455.8, -12.3, 180.88], [0.000389, 0.707107, 0.705753, -0.043742], [0,0,0,0], [9E9, 9E9, 9E9, 9E9, 9E9, 9E9]];
	VAR robtarget Openhole_3750 := [[456.25, -12.09, 180.84], [0.001203, 0.707106, 0.70561, -0.045977], [0,0,0,0], [9E9, 9E9, 9E9, 9E9, 9E9, 9E9]];
	VAR robtarget Openhole_3751 := [[456.7, -11.89, 180.8], [0.002055, 0.707104, 0.705462, -0.048195], [0,0,0,0], [9E9, 9E9, 9E9, 9E9, 9E9, 9E9]];
	VAR robtarget Openhole_3752 := [[457.17, -11.7, 180.75], [0.003016, 0.7071, 0.705311, -0.050366], [0,0,0,0], [9E9, 9E9, 9E9, 9E9, 9E9, 9E9]];
	VAR robtarget Openhole_3753 := [[458.11, -11.38, 180.66], [0.005109, 0.707088, 0.704994, -0.054621], [0,0,0,0], [9E9, 9E9, 9E9, 9E9, 9E9, 9E9]];
	VAR robtarget Openhole_3754 := [[464.29, -9.52, 179.93], [0.01985, 0.706828, 0.702416, -0.081314], [0,0,0,0], [9E9, 9E9, 9E9, 9E9, 9E9, 9E9]];
	VAR robtarget Openhole_3755 := [[464.77, -9.39, 179.87], [0.021022, 0.706794, 0.702181, -0.083314], [0,0,0,0], [9E9, 9E9, 9E9, 9E9, 9E9, 9E9]];
	VAR robtarget Openhole_3756 := [[469.61, -8.3, 179.21], [0.033606, 0.706308, 0.699638, -0.102502], [0,0,0,0], [9E9, 9E9, 9E9, 9E9, 9E9, 9E9]];
	VAR robtarget Openhole_3757 := [[474.02, -7.68, 178.61], [0.046177, 0.705597, 0.697122, -0.118413], [0,0,0,0], [9E9, 9E9, 9E9, 9E9, 9E9, 9E9]];
	VAR robtarget Openhole_3758 := [[478.47, -7.38, 178.04], [0.059751, 0.704578, 0.694492, -0.132968], [0,0,0,0], [9E9, 9E9, 9E9, 9E9, 9E9, 9E9]];
	VAR robtarget Openhole_3759 := [[480.96, -7.35, 177.75], [0.067631, 0.703865, 0.693011, -0.140482], [0,0,0,0], [9E9, 9E9, 9E9, 9E9, 9E9, 9E9]];
	VAR robtarget Openhole_3760 := [[481.45, -7.35, 177.69], [0.06922, 0.703711, 0.692713, -0.141946], [0,0,0,0], [9E9, 9E9, 9E9, 9E9, 9E9, 9E9]];
	VAR robtarget Openhole_3761 := [[487.92, -7.59, 177.06], [0.090206, 0.701329, 0.688808, -0.159822], [0,0,0,0], [9E9, 9E9, 9E9, 9E9, 9E9, 9E9]];
	VAR robtarget Openhole_3762 := [[499.86, -8.3, 176.09], [0.127581, 0.695502, 0.681203, -0.189637], [0,0,0,0], [9E9, 9E9, 9E9, 9E9, 9E9, 9E9]];
	VAR robtarget Openhole_3763 := [[501.35, -8.33, 175.94], [0.13184, 0.694707, 0.680164, -0.193332], [0,0,0,0], [9E9, 9E9, 9E9, 9E9, 9E9, 9E9]];
	VAR robtarget Openhole_3764 := [[501.85, -8.33, 175.89], [0.133222, 0.694444, 0.679809, -0.194576], [0,0,0,0], [9E9, 9E9, 9E9, 9E9, 9E9, 9E9]];
	VAR robtarget Openhole_3765 := [[503.83, -8.3, 175.68], [0.138627, 0.693385, 0.678364, -0.199556], [0,0,0,0], [9E9, 9E9, 9E9, 9E9, 9E9, 9E9]];
	VAR robtarget Openhole_3766 := [[504.35, -8.28, 175.61], [0.139966, 0.693116, 0.677966, -0.200903], [0,0,0,0], [9E9, 9E9, 9E9, 9E9, 9E9, 9E9]];
	VAR robtarget Openhole_3767 := [[509.33, -8.28, 175.09], [0.183051, 0.683002, 0.683002, -0.183051], [0,0,0,0], [9E9, 9E9, 9E9, 9E9, 9E9, 9E9]];
	VAR robtarget Openhole_3768 := [[536.33, -8.27, 175.01], [0.183051, 0.683002, 0.683002, -0.183051], [0,0,0,0], [9E9, 9E9, 9E9, 9E9, 9E9, 9E9]];
	VAR robtarget Openhole_3769 := [[536.33, -9.15, 175.51], [0.183051, 0.683002, 0.683002, -0.183051], [0,0,0,0], [9E9, 9E9, 9E9, 9E9, 9E9, 9E9]];
	VAR robtarget Openhole_3770 := [[509.33, -9.15, 175.6], [0.183051, 0.683002, 0.683002, -0.183051], [0,0,0,0], [9E9, 9E9, 9E9, 9E9, 9E9, 9E9]];
	VAR robtarget Openhole_3771 := [[504.33, -9.15, 176.07], [0.142442, 0.692611, 0.678716, -0.198353], [0,0,0,0], [9E9, 9E9, 9E9, 9E9, 9E9, 9E9]];
	VAR robtarget Openhole_3772 := [[503.69, -9.17, 176.15], [0.140778, 0.692951, 0.679197, -0.196703], [0,0,0,0], [9E9, 9E9, 9E9, 9E9, 9E9, 9E9]];
	VAR robtarget Openhole_3773 := [[503.19, -9.2, 176.21], [0.139523, 0.693205, 0.679576, -0.195388], [0,0,0,0], [9E9, 9E9, 9E9, 9E9, 9E9, 9E9]];
	VAR robtarget Openhole_3774 := [[500.21, -9.26, 176.52], [0.131436, 0.694784, 0.681729, -0.187738], [0,0,0,0], [9E9, 9E9, 9E9, 9E9, 9E9, 9E9]];
	VAR robtarget Openhole_3775 := [[499.71, -9.26, 176.56], [0.130032, 0.695048, 0.682076, -0.186474], [0,0,0,0], [9E9, 9E9, 9E9, 9E9, 9E9, 9E9]];
	VAR robtarget Openhole_3776 := [[491.74, -8.94, 177.18], [0.10599, 0.699118, 0.68727, -0.166313], [0,0,0,0], [9E9, 9E9, 9E9, 9E9, 9E9, 9E9]];
	VAR robtarget Openhole_3777 := [[482.78, -8.57, 177.93], [0.077316, 0.702867, 0.692694, -0.142038], [0,0,0,0], [9E9, 9E9, 9E9, 9E9, 9E9, 9E9]];
	VAR robtarget Openhole_3778 := [[481.79, -8.56, 178.03], [0.074151, 0.703208, 0.693285, -0.139127], [0,0,0,0], [9E9, 9E9, 9E9, 9E9, 9E9, 9E9]];
	VAR robtarget Openhole_3779 := [[481.29, -8.56, 178.08], [0.072577, 0.703372, 0.693579, -0.137651], [0,0,0,0], [9E9, 9E9, 9E9, 9E9, 9E9, 9E9]];
	VAR robtarget Openhole_3780 := [[476.32, -8.73, 178.63], [0.057153, 0.704793, 0.69648, -0.122127], [0,0,0,0], [9E9, 9E9, 9E9, 9E9, 9E9, 9E9]];
	VAR robtarget Openhole_3781 := [[471.89, -9.23, 179.18], [0.044252, 0.705721, 0.699011, -0.106695], [0,0,0,0], [9E9, 9E9, 9E9, 9E9, 9E9, 9E9]];
	VAR robtarget Openhole_3782 := [[468.97, -9.8, 179.56], [0.036434, 0.706167, 0.700621, -0.095551], [0,0,0,0], [9E9, 9E9, 9E9, 9E9, 9E9, 9E9]];
	VAR robtarget Openhole_3783 := [[466.57, -10.43, 179.88], [0.030503, 0.706449, 0.701889, -0.08574], [0,0,0,0], [9E9, 9E9, 9E9, 9E9, 9E9, 9E9]];
	VAR robtarget Openhole_3784 := [[463.74, -11.36, 180.24], [0.02415, 0.706694, 0.703289, -0.073382], [0,0,0,0], [9E9, 9E9, 9E9, 9E9, 9E9, 9E9]];
	VAR robtarget Openhole_3785 := [[461.9, -12.1, 180.46], [0.020409, 0.706812, 0.70413, -0.06482], [0,0,0,0], [9E9, 9E9, 9E9, 9E9, 9E9, 9E9]];
	VAR robtarget Openhole_3786 := [[460.54, -12.71, 180.62], [0.01784, 0.706882, 0.704703, -0.058255], [0,0,0,0], [9E9, 9E9, 9E9, 9E9, 9E9, 9E9]];
	VAR robtarget Openhole_3787 := [[459.64, -13.14, 180.72], [0.016278, 0.706919, 0.705057, -0.053804], [0,0,0,0], [9E9, 9E9, 9E9, 9E9, 9E9, 9E9]];
	VAR robtarget Openhole_3788 := [[459.2, -13.37, 180.77], [0.015555, 0.706936, 0.705225, -0.051554], [0,0,0,0], [9E9, 9E9, 9E9, 9E9, 9E9, 9E9]];
	VAR robtarget Openhole_3789 := [[458.76, -13.61, 180.81], [0.014878, 0.70695, 0.705387, -0.049286], [0,0,0,0], [9E9, 9E9, 9E9, 9E9, 9E9, 9E9]];
	VAR robtarget Openhole_3790 := [[457.91, -14.13, 180.9], [0.013724, 0.706974, 0.705693, -0.044687], [0,0,0,0], [9E9, 9E9, 9E9, 9E9, 9E9, 9E9]];
	VAR robtarget Openhole_3791 := [[456.45, -15.03, 181.03], [0.011857, 0.707007, 0.706152, -0.036732], [0,0,0,0], [9E9, 9E9, 9E9, 9E9, 9E9, 9E9]];
	VAR robtarget Openhole_3792 := [[454.01, -15.03, 181.12], [0.00354, 0.707098, 0.706534, -0.028459], [0,0,0,0], [9E9, 9E9, 9E9, 9E9, 9E9, 9E9]];
	VAR robtarget Openhole_3793 := [[454.58, -16.45, 181.17], [0.010306, 0.707032, 0.706644, -0.025565], [0,0,0,0], [9E9, 9E9, 9E9, 9E9, 9E9, 9E9]];
	VAR robtarget Openhole_3794 := [[457.02, -16.45, 181.11], [0.018611, 0.706862, 0.706297, -0.03384], [0,0,0,0], [9E9, 9E9, 9E9, 9E9, 9E9, 9E9]];
	VAR robtarget Openhole_3795 := [[457.6, -16.2, 181.08], [0.019698, 0.706832, 0.706157, -0.03664], [0,0,0,0], [9E9, 9E9, 9E9, 9E9, 9E9, 9E9]];
	VAR robtarget Openhole_3796 := [[458.48, -15.74, 181.01], [0.021141, 0.706791, 0.705907, -0.041176], [0,0,0,0], [9E9, 9E9, 9E9, 9E9, 9E9, 9E9]];
	VAR robtarget Openhole_3797 := [[458.92, -15.49, 180.98], [0.021766, 0.706772, 0.705769, -0.043468], [0,0,0,0], [9E9, 9E9, 9E9, 9E9, 9E9, 9E9]];
	VAR robtarget Openhole_3798 := [[459.34, -15.23, 180.94], [0.022319, 0.706754, 0.705624, -0.045774], [0,0,0,0], [9E9, 9E9, 9E9, 9E9, 9E9, 9E9]];
	VAR robtarget Openhole_3799 := [[460.18, -14.69, 180.85], [0.023321, 0.706722, 0.705308, -0.0504], [0,0,0,0], [9E9, 9E9, 9E9, 9E9, 9E9, 9E9]];
	VAR robtarget Openhole_3800 := [[461.04, -14.18, 180.76], [0.024495, 0.706682, 0.704967, -0.054971], [0,0,0,0], [9E9, 9E9, 9E9, 9E9, 9E9, 9E9]];
	VAR robtarget Openhole_3801 := [[463.23, -13.02, 180.5], [0.027995, 0.706552, 0.704004, -0.066168], [0,0,0,0], [9E9, 9E9, 9E9, 9E9, 9E9, 9E9]];
	VAR robtarget Openhole_3802 := [[463.68, -12.81, 180.44], [0.028797, 0.70652, 0.703795, -0.068361], [0,0,0,0], [9E9, 9E9, 9E9, 9E9, 9E9, 9E9]];
	VAR robtarget Openhole_3803 := [[465.05, -12.22, 180.27], [0.031419, 0.706408, 0.703136, -0.074829], [0,0,0,0], [9E9, 9E9, 9E9, 9E9, 9E9, 9E9]];
	VAR robtarget Openhole_3804 := [[465.51, -12.04, 180.21], [0.032363, 0.706366, 0.702908, -0.076946], [0,0,0,0], [9E9, 9E9, 9E9, 9E9, 9E9, 9E9]];
	VAR robtarget Openhole_3805 := [[468.83, -10.99, 179.79], [0.039929, 0.705979, 0.701205, -0.091165], [0,0,0,0], [9E9, 9E9, 9E9, 9E9, 9E9, 9E9]];
	VAR robtarget Openhole_3806 := [[469.79, -10.75, 179.67], [0.042336, 0.705838, 0.70069, -0.095043], [0,0,0,0], [9E9, 9E9, 9E9, 9E9, 9E9, 9E9]];
	VAR robtarget Openhole_3807 := [[473.7, -10.06, 179.2], [0.052944, 0.705122, 0.698549, -0.109681], [0,0,0,0], [9E9, 9E9, 9E9, 9E9, 9E9, 9E9]];
	VAR robtarget Openhole_3808 := [[478.16, -9.69, 178.71], [0.066189, 0.704002, 0.696034, -0.124644], [0,0,0,0], [9E9, 9E9, 9E9, 9E9, 9E9, 9E9]];
	VAR robtarget Openhole_3809 := [[482.14, -9.61, 178.33], [0.078623, 0.702722, 0.693741, -0.136831], [0,0,0,0], [9E9, 9E9, 9E9, 9E9, 9E9, 9E9]];
	VAR robtarget Openhole_3810 := [[482.64, -9.62, 178.29], [0.080197, 0.702544, 0.693451, -0.138297], [0,0,0,0], [9E9, 9E9, 9E9, 9E9, 9E9, 9E9]];
	VAR robtarget Openhole_3811 := [[494.09, -10.02, 177.42], [0.116232, 0.697488, 0.686503, -0.169449], [0,0,0,0], [9E9, 9E9, 9E9, 9E9, 9E9, 9E9]];
	VAR robtarget Openhole_3812 := [[499.58, -10.13, 177], [0.132245, 0.69463, 0.682862, -0.183576], [0,0,0,0], [9E9, 9E9, 9E9, 9E9, 9E9, 9E9]];
	VAR robtarget Openhole_3813 := [[500.08, -10.12, 176.95], [0.133631, 0.694365, 0.682515, -0.18486], [0,0,0,0], [9E9, 9E9, 9E9, 9E9, 9E9, 9E9]];
	VAR robtarget Openhole_3814 := [[503.56, -10.02, 176.6], [0.142895, 0.692518, 0.679991, -0.193937], [0,0,0,0], [9E9, 9E9, 9E9, 9E9, 9E9, 9E9]];
	VAR robtarget Openhole_3815 := [[504.33, -10, 176.53], [0.144956, 0.692089, 0.679431, -0.195891], [0,0,0,0], [9E9, 9E9, 9E9, 9E9, 9E9, 9E9]];
	VAR robtarget Openhole_3816 := [[509.33, -10, 176.09], [0.183051, 0.683002, 0.683002, -0.183051], [0,0,0,0], [9E9, 9E9, 9E9, 9E9, 9E9, 9E9]];
	VAR robtarget Openhole_3817 := [[536.33, -10, 176.01], [0.183051, 0.683002, 0.683002, -0.183051], [0,0,0,0], [9E9, 9E9, 9E9, 9E9, 9E9, 9E9]];
	VAR robtarget Openhole_3818 := [[536.33, -10.89, 176.52], [0.183051, 0.683002, 0.683002, -0.183051], [0,0,0,0], [9E9, 9E9, 9E9, 9E9, 9E9, 9E9]];
	VAR robtarget Openhole_3819 := [[524.33, -10.89, 176.55], [0.183051, 0.683002, 0.683002, -0.183051], [0,0,0,0], [9E9, 9E9, 9E9, 9E9, 9E9, 9E9]];
	VAR robtarget Openhole_3820 := [[509.33, -10.89, 176.6], [0.183051, 0.683002, 0.683002, -0.183051], [0,0,0,0], [9E9, 9E9, 9E9, 9E9, 9E9, 9E9]];
	VAR robtarget Openhole_3821 := [[504.39, -10.89, 176.99], [0.147705, 0.691508, 0.680116, -0.193501], [0,0,0,0], [9E9, 9E9, 9E9, 9E9, 9E9, 9E9]];
	VAR robtarget Openhole_3822 := [[498.87, -11.14, 177.54], [0.133281, 0.694432, 0.684139, -0.178758], [0,0,0,0], [9E9, 9E9, 9E9, 9E9, 9E9, 9E9]];
	VAR robtarget Openhole_3823 := [[497.37, -11.14, 177.66], [0.129086, 0.695224, 0.685156, -0.174817], [0,0,0,0], [9E9, 9E9, 9E9, 9E9, 9E9, 9E9]];
	VAR robtarget Openhole_3824 := [[496.87, -11.14, 177.69], [0.127662, 0.695487, 0.685489, -0.173507], [0,0,0,0], [9E9, 9E9, 9E9, 9E9, 9E9, 9E9]];
	VAR robtarget Openhole_3825 := [[482.41, -10.79, 178.68], [0.083264, 0.702187, 0.694311, -0.13391], [0,0,0,0], [9E9, 9E9, 9E9, 9E9, 9E9, 9E9]];
	VAR robtarget Openhole_3826 := [[481.91, -10.8, 178.72], [0.081702, 0.702371, 0.694596, -0.132425], [0,0,0,0], [9E9, 9E9, 9E9, 9E9, 9E9, 9E9]];
	VAR robtarget Openhole_3827 := [[476.44, -10.97, 179.2], [0.064808, 0.704131, 0.69765, -0.115261], [0,0,0,0], [9E9, 9E9, 9E9, 9E9, 9E9, 9E9]];
	VAR robtarget Openhole_3828 := [[472.49, -11.44, 179.61], [0.053485, 0.705081, 0.6998, -0.101393], [0,0,0,0], [9E9, 9E9, 9E9, 9E9, 9E9, 9E9]];
	VAR robtarget Openhole_3829 := [[471.02, -11.7, 179.77], [0.049521, 0.705371, 0.700577, -0.095873], [0,0,0,0], [9E9, 9E9, 9E9, 9E9, 9E9, 9E9]];
	VAR robtarget Openhole_3830 := [[470.53, -11.8, 179.83], [0.048255, 0.705458, 0.700833, -0.093985], [0,0,0,0], [9E9, 9E9, 9E9, 9E9, 9E9, 9E9]];
	VAR robtarget Openhole_3831 := [[469.57, -12.03, 179.94], [0.045816, 0.705621, 0.701339, -0.090132], [0,0,0,0], [9E9, 9E9, 9E9, 9E9, 9E9, 9E9]];
	VAR robtarget Openhole_3832 := [[468.61, -12.29, 180.05], [0.043501, 0.705767, 0.701835, -0.086183], [0,0,0,0], [9E9, 9E9, 9E9, 9E9, 9E9, 9E9]];
	VAR robtarget Openhole_3833 := [[467.66, -12.58, 180.16], [0.041312, 0.705899, 0.702319, -0.082142], [0,0,0,0], [9E9, 9E9, 9E9, 9E9, 9E9, 9E9]];
	VAR robtarget Openhole_3834 := [[466.25, -13.07, 180.33], [0.038288, 0.706069, 0.70302, -0.075913], [0,0,0,0], [9E9, 9E9, 9E9, 9E9, 9E9, 9E9]];
	VAR robtarget Openhole_3835 := [[465.79, -13.26, 180.39], [0.037363, 0.706119, 0.703246, -0.073789], [0,0,0,0], [9E9, 9E9, 9E9, 9E9, 9E9, 9E9]];
	VAR robtarget Openhole_3836 := [[465.33, -13.45, 180.44], [0.036484, 0.706165, 0.703468, -0.071641], [0,0,0,0], [9E9, 9E9, 9E9, 9E9, 9E9, 9E9]];
	VAR robtarget Openhole_3837 := [[464.88, -13.66, 180.5], [0.035662, 0.706207, 0.703686, -0.069467], [0,0,0,0], [9E9, 9E9, 9E9, 9E9, 9E9, 9E9]];
	VAR robtarget Openhole_3838 := [[463.11, -14.56, 180.71], [0.032767, 0.706347, 0.704506, -0.060588], [0,0,0,0], [9E9, 9E9, 9E9, 9E9, 9E9, 9E9]];
	VAR robtarget Openhole_3839 := [[461.82, -15.31, 180.86], [0.030959, 0.706429, 0.705059, -0.053777], [0,0,0,0], [9E9, 9E9, 9E9, 9E9, 9E9, 9E9]];
	VAR robtarget Openhole_3840 := [[460.15, -16.4, 181.03], [0.029002, 0.706512, 0.705703, -0.044533], [0,0,0,0], [9E9, 9E9, 9E9, 9E9, 9E9, 9E9]];
	VAR robtarget Openhole_3841 := [[459.72, -16.65, 181.06], [0.028409, 0.706536, 0.705844, -0.042237], [0,0,0,0], [9E9, 9E9, 9E9, 9E9, 9E9, 9E9]];
	VAR robtarget Openhole_3842 := [[459.27, -16.88, 181.1], [0.027653, 0.706566, 0.705975, -0.039985], [0,0,0,0], [9E9, 9E9, 9E9, 9E9, 9E9, 9E9]];
	VAR robtarget Openhole_3843 := [[458.82, -17.08, 181.12], [0.026805, 0.706599, 0.706098, -0.037763], [0,0,0,0], [9E9, 9E9, 9E9, 9E9, 9E9, 9E9]];
	VAR robtarget Openhole_3844 := [[458.35, -17.26, 181.15], [0.02585, 0.706634, 0.706211, -0.035581], [0,0,0,0], [9E9, 9E9, 9E9, 9E9, 9E9, 9E9]];
	VAR robtarget Openhole_3845 := [[457.88, -17.43, 181.17], [0.024838, 0.70667, 0.706316, -0.033423], [0,0,0,0], [9E9, 9E9, 9E9, 9E9, 9E9, 9E9]];
	VAR robtarget Openhole_3846 := [[457.27, -17.6, 181.19], [0.02333, 0.706722, 0.706436, -0.030789], [0,0,0,0], [9E9, 9E9, 9E9, 9E9, 9E9, 9E9]];
	VAR robtarget Openhole_3847 := [[454.82, -17.6, 181.23], [0.015035, 0.706947, 0.706748, -0.022509], [0,0,0,0], [9E9, 9E9, 9E9, 9E9, 9E9, 9E9]];
	VAR robtarget Openhole_3848 := [[454.9, -18.58, 181.28], [0.018612, 0.706862, 0.706839, -0.019447], [0,0,0,0], [9E9, 9E9, 9E9, 9E9, 9E9, 9E9]];
	VAR robtarget Openhole_3849 := [[457.35, -18.58, 181.27], [0.0269, 0.706595, 0.706563, -0.027733], [0,0,0,0], [9E9, 9E9, 9E9, 9E9, 9E9, 9E9]];
	VAR robtarget Openhole_3850 := [[457.46, -18.57, 181.27], [0.027297, 0.70658, 0.706547, -0.028138], [0,0,0,0], [9E9, 9E9, 9E9, 9E9, 9E9, 9E9]];
	VAR robtarget Openhole_3851 := [[457.96, -18.57, 181.26], [0.02897, 0.706513, 0.706477, -0.029843], [0,0,0,0], [9E9, 9E9, 9E9, 9E9, 9E9, 9E9]];
	VAR robtarget Openhole_3852 := [[458.45, -18.46, 181.25], [0.030247, 0.70646, 0.706389, -0.031858], [0,0,0,0], [9E9, 9E9, 9E9, 9E9, 9E9, 9E9]];
	VAR robtarget Openhole_3853 := [[459.42, -18.22, 181.22], [0.03269, 0.706351, 0.706192, -0.035949], [0,0,0,0], [9E9, 9E9, 9E9, 9E9, 9E9, 9E9]];
	VAR robtarget Openhole_3854 := [[460.37, -17.92, 181.18], [0.034892, 0.706245, 0.705965, -0.040162], [0,0,0,0], [9E9, 9E9, 9E9, 9E9, 9E9, 9E9]];
	VAR robtarget Openhole_3855 := [[460.84, -17.74, 181.16], [0.035843, 0.706198, 0.705838, -0.042335], [0,0,0,0], [9E9, 9E9, 9E9, 9E9, 9E9, 9E9]];
	VAR robtarget Openhole_3856 := [[461.3, -17.54, 181.13], [0.036739, 0.706152, 0.705703, -0.044529], [0,0,0,0], [9E9, 9E9, 9E9, 9E9, 9E9, 9E9]];
	VAR robtarget Openhole_3857 := [[462.19, -17.09, 181.06], [0.038176, 0.706076, 0.705405, -0.049032], [0,0,0,0], [9E9, 9E9, 9E9, 9E9, 9E9, 9E9]];
	VAR robtarget Openhole_3858 := [[463.94, -16.14, 180.9], [0.040871, 0.705925, 0.70472, -0.058046], [0,0,0,0], [9E9, 9E9, 9E9, 9E9, 9E9, 9E9]];
	VAR robtarget Openhole_3859 := [[464.83, -15.7, 180.81], [0.04234, 0.705838, 0.70434, -0.06249], [0,0,0,0], [9E9, 9E9, 9E9, 9E9, 9E9, 9E9]];
	VAR robtarget Openhole_3860 := [[465.73, -15.28, 180.71], [0.043936, 0.70574, 0.703938, -0.066871], [0,0,0,0], [9E9, 9E9, 9E9, 9E9, 9E9, 9E9]];
	VAR robtarget Openhole_3861 := [[466.19, -15.08, 180.66], [0.044792, 0.705687, 0.703729, -0.069033], [0,0,0,0], [9E9, 9E9, 9E9, 9E9, 9E9, 9E9]];
	VAR robtarget Openhole_3862 := [[466.65, -14.89, 180.61], [0.045688, 0.705629, 0.703516, -0.071174], [0,0,0,0], [9E9, 9E9, 9E9, 9E9, 9E9, 9E9]];
	VAR robtarget Openhole_3863 := [[467.12, -14.71, 180.56], [0.046638, 0.705567, 0.703299, -0.073287], [0,0,0,0], [9E9, 9E9, 9E9, 9E9, 9E9, 9E9]];
	VAR robtarget Openhole_3864 := [[467.59, -14.54, 180.51], [0.047636, 0.7055, 0.703078, -0.075373], [0,0,0,0], [9E9, 9E9, 9E9, 9E9, 9E9, 9E9]];
	VAR robtarget Openhole_3865 := [[468.53, -14.24, 180.42], [0.049753, 0.705354, 0.702627, -0.079469], [0,0,0,0], [9E9, 9E9, 9E9, 9E9, 9E9, 9E9]];
	VAR robtarget Openhole_3866 := [[469.49, -13.97, 180.32], [0.052017, 0.705191, 0.702163, -0.083468], [0,0,0,0], [9E9, 9E9, 9E9, 9E9, 9E9, 9E9]];
	VAR robtarget Openhole_3867 := [[470.46, -13.73, 180.22], [0.054392, 0.705012, 0.701687, -0.087379], [0,0,0,0], [9E9, 9E9, 9E9, 9E9, 9E9, 9E9]];
	VAR robtarget Openhole_3868 := [[470.94, -13.62, 180.18], [0.055622, 0.704916, 0.701445, -0.089299], [0,0,0,0], [9E9, 9E9, 9E9, 9E9, 9E9, 9E9]];
	VAR robtarget Openhole_3869 := [[471.92, -13.42, 180.08], [0.058168, 0.70471, 0.700955, -0.093069], [0,0,0,0], [9E9, 9E9, 9E9, 9E9, 9E9, 9E9]];
	VAR robtarget Openhole_3870 := [[475.87, -12.91, 179.74], [0.069332, 0.7037, 0.698936, -0.107185], [0,0,0,0], [9E9, 9E9, 9E9, 9E9, 9E9, 9E9]];
	VAR robtarget Openhole_3871 := [[480.85, -12.71, 179.39], [0.084529, 0.702036, 0.696304, -0.12313], [0,0,0,0], [9E9, 9E9, 9E9, 9E9, 9E9, 9E9]];
	VAR robtarget Openhole_3872 := [[482.35, -12.7, 179.29], [0.08918, 0.701461, 0.695487, -0.127663], [0,0,0,0], [9E9, 9E9, 9E9, 9E9, 9E9, 9E9]];
	VAR robtarget Openhole_3873 := [[482.85, -12.7, 179.26], [0.090734, 0.701261, 0.695212, -0.129152], [0,0,0,0], [9E9, 9E9, 9E9, 9E9, 9E9, 9E9]];
	VAR robtarget Openhole_3874 := [[495.33, -12.89, 178.59], [0.128579, 0.695318, 0.687801, -0.164101], [0,0,0,0], [9E9, 9E9, 9E9, 9E9, 9E9, 9E9]];
	VAR robtarget Openhole_3875 := [[495.83, -12.89, 178.56], [0.13, 0.695054, 0.687477, -0.165453], [0,0,0,0], [9E9, 9E9, 9E9, 9E9, 9E9, 9E9]];
	VAR robtarget Openhole_3876 := [[501.81, -12.75, 178.13], [0.146208, 0.691826, 0.683391, -0.181596], [0,0,0,0], [9E9, 9E9, 9E9, 9E9, 9E9, 9E9]];
	VAR robtarget Openhole_3877 := [[504.34, -12.58, 177.89], [0.152514, 0.690463, 0.68153, -0.188461], [0,0,0,0], [9E9, 9E9, 9E9, 9E9, 9E9, 9E9]];
	VAR robtarget Openhole_3878 := [[509.33, -12.58, 177.58], [0.183051, 0.683002, 0.683002, -0.183051], [0,0,0,0], [9E9, 9E9, 9E9, 9E9, 9E9, 9E9]];
	VAR robtarget Openhole_3879 := [[536.33, -12.58, 177.5], [0.183051, 0.683002, 0.683002, -0.183051], [0,0,0,0], [9E9, 9E9, 9E9, 9E9, 9E9, 9E9]];
	VAR robtarget Openhole_3880 := [[536.34, -16.49, 179.75], [0.183051, 0.683002, 0.683002, -0.183051], [0,0,0,0], [9E9, 9E9, 9E9, 9E9, 9E9, 9E9]];
	VAR robtarget Openhole_3881 := [[509.34, -16.49, 179.84], [0.183051, 0.683002, 0.683002, -0.183051], [0,0,0,0], [9E9, 9E9, 9E9, 9E9, 9E9, 9E9]];
	VAR robtarget Openhole_3882 := [[504.34, -16.49, 179.96], [0.163963, 0.687834, 0.684562, -0.177129], [0,0,0,0], [9E9, 9E9, 9E9, 9E9, 9E9, 9E9]];
	VAR robtarget Openhole_3883 := [[497.74, -16.81, 180.27], [0.147217, 0.691612, 0.689035, -0.158842], [0,0,0,0], [9E9, 9E9, 9E9, 9E9, 9E9, 9E9]];
	VAR robtarget Openhole_3884 := [[491.75, -16.89, 180.43], [0.130573, 0.694947, 0.692711, -0.141954], [0,0,0,0], [9E9, 9E9, 9E9, 9E9, 9E9, 9E9]];
	VAR robtarget Openhole_3885 := [[491.25, -16.89, 180.44], [0.129129, 0.695216, 0.693001, -0.140532], [0,0,0,0], [9E9, 9E9, 9E9, 9E9, 9E9, 9E9]];
	VAR robtarget Openhole_3886 := [[478.25, -16.73, 180.66], [0.08936, 0.701438, 0.699684, -0.10219], [0,0,0,0], [9E9, 9E9, 9E9, 9E9, 9E9, 9E9]];
	VAR robtarget Openhole_3887 := [[477.75, -16.74, 180.68], [0.087791, 0.701636, 0.69991, -0.100628], [0,0,0,0], [9E9, 9E9, 9E9, 9E9, 9E9, 9E9]];
	VAR robtarget Openhole_3888 := [[472.25, -16.88, 180.83], [0.070685, 0.703565, 0.702248, -0.082754], [0,0,0,0], [9E9, 9E9, 9E9, 9E9, 9E9, 9E9]];
	VAR robtarget Openhole_3889 := [[471.26, -16.95, 180.86], [0.067703, 0.703858, 0.702647, -0.079294], [0,0,0,0], [9E9, 9E9, 9E9, 9E9, 9E9, 9E9]];
	VAR robtarget Openhole_3890 := [[470.26, -17.06, 180.91], [0.064832, 0.704128, 0.703041, -0.075717], [0,0,0,0], [9E9, 9E9, 9E9, 9E9, 9E9, 9E9]];
	VAR robtarget Openhole_3891 := [[468.29, -17.35, 181], [0.059324, 0.704614, 0.703799, -0.068311], [0,0,0,0], [9E9, 9E9, 9E9, 9E9, 9E9, 9E9]];
	VAR robtarget Openhole_3892 := [[467.8, -17.44, 181.02], [0.058006, 0.704724, 0.703982, -0.066404], [0,0,0,0], [9E9, 9E9, 9E9, 9E9, 9E9, 9E9]];
	VAR robtarget Openhole_3893 := [[467.31, -17.54, 181.04], [0.056726, 0.704828, 0.704162, -0.064465], [0,0,0,0], [9E9, 9E9, 9E9, 9E9, 9E9, 9E9]];
	VAR robtarget Openhole_3894 := [[465.37, -18.02, 181.15], [0.051899, 0.7052, 0.704848, -0.056477], [0,0,0,0], [9E9, 9E9, 9E9, 9E9, 9E9, 9E9]];
	VAR robtarget Openhole_3895 := [[464.4, -18.28, 181.19], [0.049599, 0.705365, 0.705163, -0.052389], [0,0,0,0], [9E9, 9E9, 9E9, 9E9, 9E9, 9E9]];
	VAR robtarget Openhole_3896 := [[463.43, -18.53, 181.23], [0.047197, 0.70553, 0.705452, -0.048342], [0,0,0,0], [9E9, 9E9, 9E9, 9E9, 9E9, 9E9]];
	VAR robtarget Openhole_3897 := [[460.01, -19.25, 181.32], [0.03817, 0.706076, 0.706268, -0.034441], [0,0,0,0], [9E9, 9E9, 9E9, 9E9, 9E9, 9E9]];
	VAR robtarget Openhole_3898 := [[458.04, -19.56, 181.35], [0.032567, 0.706356, 0.706601, -0.02673], [0,0,0,0], [9E9, 9E9, 9E9, 9E9, 9E9, 9E9]];
	VAR robtarget Openhole_3899 := [[457.29, -19.61, 181.35], [0.030238, 0.70646, 0.706698, -0.024052], [0,0,0,0], [9E9, 9E9, 9E9, 9E9, 9E9, 9E9]];
	VAR robtarget Openhole_3900 := [[454.85, -19.61, 181.33], [0.021956, 0.706766, 0.706931, -0.015759], [0,0,0,0], [9E9, 9E9, 9E9, 9E9, 9E9, 9E9]];
	VAR robtarget Openhole_3901 := [[454.66, -20.66, 181.38], [0.024872, 0.706669, 0.707013, -0.011543], [0,0,0,0], [9E9, 9E9, 9E9, 9E9, 9E9, 9E9]];
	VAR robtarget Openhole_3902 := [[457.1, -20.66, 181.42], [0.03315, 0.706329, 0.706828, -0.019844], [0,0,0,0], [9E9, 9E9, 9E9, 9E9, 9E9, 9E9]];
	VAR robtarget Openhole_3903 := [[457.64, -20.63, 181.43], [0.034885, 0.706246, 0.706772, -0.021772], [0,0,0,0], [9E9, 9E9, 9E9, 9E9, 9E9, 9E9]];
	VAR robtarget Openhole_3904 := [[458.63, -20.47, 181.43], [0.037651, 0.706104, 0.706641, -0.025665], [0,0,0,0], [9E9, 9E9, 9E9, 9E9, 9E9, 9E9]];
	VAR robtarget Openhole_3905 := [[459.13, -20.43, 181.43], [0.039189, 0.70602, 0.706572, -0.027486], [0,0,0,0], [9E9, 9E9, 9E9, 9E9, 9E9, 9E9]];
	VAR robtarget Openhole_3906 := [[460.13, -20.37, 181.44], [0.042353, 0.705837, 0.706425, -0.031041], [0,0,0,0], [9E9, 9E9, 9E9, 9E9, 9E9, 9E9]];
	VAR robtarget Openhole_3907 := [[461.63, -20.35, 181.46], [0.047297, 0.705523, 0.706181, -0.036163], [0,0,0,0], [9E9, 9E9, 9E9, 9E9, 9E9, 9E9]];
	VAR robtarget Openhole_3908 := [[462.63, -20.37, 181.47], [0.050686, 0.705288, 0.706005, -0.039462], [0,0,0,0], [9E9, 9E9, 9E9, 9E9, 9E9, 9E9]];
	VAR robtarget Openhole_3909 := [[464.13, -20.42, 181.5], [0.055867, 0.704896, 0.705719, -0.044272], [0,0,0,0], [9E9, 9E9, 9E9, 9E9, 9E9, 9E9]];
	VAR robtarget Openhole_3910 := [[480.61, -20.9, 181.87], [0.11018, 0.69847, 0.700551, -0.096064], [0,0,0,0], [9E9, 9E9, 9E9, 9E9, 9E9, 9E9]];
	VAR robtarget Openhole_3911 := [[489.11, -20.98, 182.05], [0.135699, 0.693964, 0.696574, -0.12159], [0,0,0,0], [9E9, 9E9, 9E9, 9E9, 9E9, 9E9]];
	VAR robtarget Openhole_3912 := [[489.61, -20.98, 182.06], [0.137135, 0.693681, 0.696315, -0.123065], [0,0,0,0], [9E9, 9E9, 9E9, 9E9, 9E9, 9E9]];
	VAR robtarget Openhole_3913 := [[499.61, -20.8, 182.16], [0.164227, 0.687771, 0.690593, -0.151924], [0,0,0,0], [9E9, 9E9, 9E9, 9E9, 9E9, 9E9]];
	VAR robtarget Openhole_3914 := [[504.35, -20.6, 182.13], [0.175939, 0.684869, 0.687545, -0.165174], [0,0,0,0], [9E9, 9E9, 9E9, 9E9, 9E9, 9E9]];
	VAR robtarget Openhole_3915 := [[509.35, -20.6, 182.21], [0.183051, 0.683002, 0.683002, -0.183051], [0,0,0,0], [9E9, 9E9, 9E9, 9E9, 9E9, 9E9]];
	VAR robtarget Openhole_3916 := [[536.35, -20.6, 182.12], [0.183051, 0.683002, 0.683002, -0.183051], [0,0,0,0], [9E9, 9E9, 9E9, 9E9, 9E9, 9E9]];
	VAR robtarget Openhole_3917 := [[536.35, -22.17, 183.03], [0.183051, 0.683002, 0.683002, -0.183051], [0,0,0,0], [9E9, 9E9, 9E9, 9E9, 9E9, 9E9]];
	VAR robtarget Openhole_3918 := [[509.35, -22.17, 183.12], [0.183051, 0.683002, 0.683002, -0.183051], [0,0,0,0], [9E9, 9E9, 9E9, 9E9, 9E9, 9E9]];
	VAR robtarget Openhole_3919 := [[504.35, -22.17, 182.96], [0.180517, 0.683677, 0.688633, -0.160577], [0,0,0,0], [9E9, 9E9, 9E9, 9E9, 9E9, 9E9]];
	VAR robtarget Openhole_3920 := [[494.58, -22.52, 182.82], [0.155823, 0.689724, 0.694545, -0.13269], [0,0,0,0], [9E9, 9E9, 9E9, 9E9, 9E9, 9E9]];
	VAR robtarget Openhole_3921 := [[485.58, -22.61, 182.55], [0.130521, 0.694956, 0.699133, -0.105889], [0,0,0,0], [9E9, 9E9, 9E9, 9E9, 9E9, 9E9]];
	VAR robtarget Openhole_3922 := [[485.08, -22.61, 182.53], [0.129049, 0.695231, 0.699362, -0.104368], [0,0,0,0], [9E9, 9E9, 9E9, 9E9, 9E9, 9E9]];
	VAR robtarget Openhole_3923 := [[471.59, -22.42, 182.03], [0.086869, 0.70175, 0.704358, -0.062293], [0,0,0,0], [9E9, 9E9, 9E9, 9E9, 9E9, 9E9]];
	VAR robtarget Openhole_3924 := [[465.61, -22.1, 181.78], [0.066372, 0.703985, 0.705761, -0.043602], [0,0,0,0], [9E9, 9E9, 9E9, 9E9, 9E9, 9E9]];
	VAR robtarget Openhole_3925 := [[461.64, -21.66, 181.61], [0.051747, 0.705211, 0.706393, -0.031771], [0,0,0,0], [9E9, 9E9, 9E9, 9E9, 9E9, 9E9]];
	VAR robtarget Openhole_3926 := [[460.14, -21.53, 181.56], [0.046326, 0.705588, 0.706585, -0.02717], [0,0,0,0], [9E9, 9E9, 9E9, 9E9, 9E9, 9E9]];
	VAR robtarget Openhole_3927 := [[459.64, -21.51, 181.55], [0.044565, 0.705701, 0.706644, -0.025574], [0,0,0,0], [9E9, 9E9, 9E9, 9E9, 9E9, 9E9]];
	VAR robtarget Openhole_3928 := [[459.14, -21.49, 181.53], [0.042847, 0.705807, 0.706702, -0.023927], [0,0,0,0], [9E9, 9E9, 9E9, 9E9, 9E9, 9E9]];
	VAR robtarget Openhole_3929 := [[458.64, -21.5, 181.52], [0.041171, 0.705907, 0.706757, -0.022234], [0,0,0,0], [9E9, 9E9, 9E9, 9E9, 9E9, 9E9]];
	VAR robtarget Openhole_3930 := [[458.15, -21.51, 181.51], [0.039546, 0.706, 0.70681, -0.020489], [0,0,0,0], [9E9, 9E9, 9E9, 9E9, 9E9, 9E9]];
	VAR robtarget Openhole_3931 := [[457.66, -21.63, 181.51], [0.038309, 0.706068, 0.706866, -0.018445], [0,0,0,0], [9E9, 9E9, 9E9, 9E9, 9E9, 9E9]];
	VAR robtarget Openhole_3932 := [[456.8, -21.6, 181.49], [0.03533, 0.706224, 0.706934, -0.015623], [0,0,0,0], [9E9, 9E9, 9E9, 9E9, 9E9, 9E9]];
	VAR robtarget Openhole_3933 := [[454.35, -21.6, 181.43], [0.027054, 0.706589, 0.707069, -0.007314], [0,0,0,0], [9E9, 9E9, 9E9, 9E9, 9E9, 9E9]];
	VAR robtarget Openhole_3934 := [[453.91, -22.56, 181.46], [0.028779, 0.706521, 0.707102, -0.002568], [0,0,0,0], [9E9, 9E9, 9E9, 9E9, 9E9, 9E9]];
	VAR robtarget Openhole_3935 := [[456.36, -22.56, 181.54], [0.037055, 0.706135, 0.707023, -0.010884], [0,0,0,0], [9E9, 9E9, 9E9, 9E9, 9E9, 9E9]];
	VAR robtarget Openhole_3936 := [[456.89, -22.57, 181.56], [0.038923, 0.706035, 0.706994, -0.012656], [0,0,0,0], [9E9, 9E9, 9E9, 9E9, 9E9, 9E9]];
	VAR robtarget Openhole_3937 := [[457.39, -22.58, 181.58], [0.040621, 0.705939, 0.706961, -0.014336], [0,0,0,0], [9E9, 9E9, 9E9, 9E9, 9E9, 9E9]];
	VAR robtarget Openhole_3938 := [[458.89, -22.62, 181.63], [0.04581, 0.705621, 0.706844, -0.019258], [0,0,0,0], [9E9, 9E9, 9E9, 9E9, 9E9, 9E9]];
	VAR robtarget Openhole_3939 := [[459.89, -22.67, 181.67], [0.049329, 0.705384, 0.70675, -0.022456], [0,0,0,0], [9E9, 9E9, 9E9, 9E9, 9E9, 9E9]];
	VAR robtarget Openhole_3940 := [[465.84, -23.34, 181.99], [0.071278, 0.703505, 0.705961, -0.040238], [0,0,0,0], [9E9, 9E9, 9E9, 9E9, 9E9, 9E9]];
	VAR robtarget Openhole_3941 := [[472.83, -23.6, 182.34], [0.094689, 0.700738, 0.704346, -0.062419], [0,0,0,0], [9E9, 9E9, 9E9, 9E9, 9E9, 9E9]];
	VAR robtarget Openhole_3942 := [[480.32, -23.66, 182.68], [0.118135, 0.697169, 0.701827, -0.086248], [0,0,0,0], [9E9, 9E9, 9E9, 9E9, 9E9, 9E9]];
	VAR robtarget Openhole_3943 := [[480.82, -23.66, 182.7], [0.119648, 0.696911, 0.701632, -0.087817], [0,0,0,0], [9E9, 9E9, 9E9, 9E9, 9E9, 9E9]];
	VAR robtarget Openhole_3944 := [[481.32, -23.66, 182.73], [0.121156, 0.69665, 0.701435, -0.089383], [0,0,0,0], [9E9, 9E9, 9E9, 9E9, 9E9, 9E9]];
	VAR robtarget Openhole_3945 := [[481.82, -23.66, 182.75], [0.122656, 0.696387, 0.701234, -0.090947], [0,0,0,0], [9E9, 9E9, 9E9, 9E9, 9E9, 9E9]];
	VAR robtarget Openhole_3946 := [[495.81, -23.48, 183.29], [0.162067, 0.688284, 0.694435, -0.133267], [0,0,0,0], [9E9, 9E9, 9E9, 9E9, 9E9, 9E9]];
	VAR robtarget Openhole_3947 := [[504.35, -23.14, 183.48], [0.183329, 0.682928, 0.689287, -0.157745], [0,0,0,0], [9E9, 9E9, 9E9, 9E9, 9E9, 9E9]];
	VAR robtarget Openhole_3948 := [[509.35, -23.14, 183.68], [0.183051, 0.683002, 0.683002, -0.183051], [0,0,0,0], [9E9, 9E9, 9E9, 9E9, 9E9, 9E9]];
	VAR robtarget Openhole_3949 := [[536.35, -23.14, 183.59], [0.183051, 0.683002, 0.683002, -0.183051], [0,0,0,0], [9E9, 9E9, 9E9, 9E9, 9E9, 9E9]];
	VAR robtarget Openhole_3950 := [[536.36, -24.03, 184.11], [0.183051, 0.683002, 0.683002, -0.183051], [0,0,0,0], [9E9, 9E9, 9E9, 9E9, 9E9, 9E9]];
	VAR robtarget Openhole_3951 := [[509.36, -24.03, 184.19], [0.183051, 0.683002, 0.683002, -0.183051], [0,0,0,0], [9E9, 9E9, 9E9, 9E9, 9E9, 9E9]];
	VAR robtarget Openhole_3952 := [[504.35, -24.03, 183.95], [0.185922, 0.682226, 0.689881, -0.155128], [0,0,0,0], [9E9, 9E9, 9E9, 9E9, 9E9, 9E9]];
	VAR robtarget Openhole_3953 := [[493.5, -24.43, 183.6], [0.158662, 0.689077, 0.696199, -0.123723], [0,0,0,0], [9E9, 9E9, 9E9, 9E9, 9E9, 9E9]];
	VAR robtarget Openhole_3954 := [[477.02, -24.66, 182.8], [0.111262, 0.698298, 0.703381, -0.072495], [0,0,0,0], [9E9, 9E9, 9E9, 9E9, 9E9, 9E9]];
	VAR robtarget Openhole_3955 := [[473.03, -24.68, 182.59], [0.098834, 0.700166, 0.704598, -0.059512], [0,0,0,0], [9E9, 9E9, 9E9, 9E9, 9E9, 9E9]];
	VAR robtarget Openhole_3956 := [[472.53, -24.68, 182.56], [0.097253, 0.700387, 0.704734, -0.057882], [0,0,0,0], [9E9, 9E9, 9E9, 9E9, 9E9, 9E9]];
	VAR robtarget Openhole_3957 := [[465.04, -24.53, 182.13], [0.07262, 0.703368, 0.70631, -0.03356], [0,0,0,0], [9E9, 9E9, 9E9, 9E9, 9E9, 9E9]];
	VAR robtarget Openhole_3958 := [[458.58, -23.97, 181.74], [0.049304, 0.705386, 0.706975, -0.013635], [0,0,0,0], [9E9, 9E9, 9E9, 9E9, 9E9, 9E9]];
	VAR robtarget Openhole_3959 := [[457.08, -23.91, 181.66], [0.044073, 0.705732, 0.707053, -0.008761], [0,0,0,0], [9E9, 9E9, 9E9, 9E9, 9E9, 9E9]];
	VAR robtarget Openhole_3960 := [[456.08, -23.86, 181.61], [0.040544, 0.705943, 0.707085, -0.005542], [0,0,0,0], [9E9, 9E9, 9E9, 9E9, 9E9, 9E9]];
	VAR robtarget Openhole_3961 := [[455.52, -23.79, 181.58], [0.038403, 0.706063, 0.707096, -0.003887], [0,0,0,0], [9E9, 9E9, 9E9, 9E9, 9E9, 9E9]];
	VAR robtarget Openhole_3962 := [[453.08, -23.79, 181.47], [0.030123, 0.706465, 0.707093, 0.004439], [0,0,0,0], [9E9, 9E9, 9E9, 9E9, 9E9, 9E9]];
	VAR robtarget Openhole_3963 := [[451.65, -25.14, 181.44], [0.029869, 0.706476, 0.706971, 0.013873], [0,0,0,0], [9E9, 9E9, 9E9, 9E9, 9E9, 9E9]];
	VAR robtarget Openhole_3964 := [[454.1, -25.14, 181.58], [0.038161, 0.706076, 0.707085, 0.005541], [0,0,0,0], [9E9, 9E9, 9E9, 9E9, 9E9, 9E9]];
	VAR robtarget Openhole_3965 := [[454.69, -25.32, 181.62], [0.040773, 0.70593, 0.707095, 0.004162], [0,0,0,0], [9E9, 9E9, 9E9, 9E9, 9E9, 9E9]];
	VAR robtarget Openhole_3966 := [[455.18, -25.38, 181.66], [0.042628, 0.705821, 0.707102, 0.002654], [0,0,0,0], [9E9, 9E9, 9E9, 9E9, 9E9, 9E9]];
	VAR robtarget Openhole_3967 := [[455.68, -25.42, 181.69], [0.04445, 0.705708, 0.707106, 0.00111], [0,0,0,0], [9E9, 9E9, 9E9, 9E9, 9E9, 9E9]];
	VAR robtarget Openhole_3968 := [[465.15, -25.83, 182.34], [0.077308, 0.702868, 0.706489, -0.029556], [0,0,0,0], [9E9, 9E9, 9E9, 9E9, 9E9, 9E9]];
	VAR robtarget Openhole_3969 := [[467.64, -25.85, 182.5], [0.085495, 0.701919, 0.706094, -0.037828], [0,0,0,0], [9E9, 9E9, 9E9, 9E9, 9E9, 9E9]];
	VAR robtarget Openhole_3970 := [[468.14, -25.85, 182.54], [0.087103, 0.701721, 0.706003, -0.039495], [0,0,0,0], [9E9, 9E9, 9E9, 9E9, 9E9, 9E9]];
	VAR robtarget Openhole_3971 := [[491.1, -25.41, 183.87], [0.155029, 0.689903, 0.697916, -0.113637], [0,0,0,0], [9E9, 9E9, 9E9, 9E9, 9E9, 9E9]];
	VAR robtarget Openhole_3972 := [[502.58, -25, 184.36], [0.184284, 0.682671, 0.691552, -0.147496], [0,0,0,0], [9E9, 9E9, 9E9, 9E9, 9E9, 9E9]];
	VAR robtarget Openhole_3973 := [[504.36, -24.92, 184.42], [0.18849, 0.681522, 0.690459, -0.152533], [0,0,0,0], [9E9, 9E9, 9E9, 9E9, 9E9, 9E9]];
	VAR robtarget Openhole_3974 := [[509.36, -24.92, 184.7], [0.183051, 0.683002, 0.683002, -0.183051], [0,0,0,0], [9E9, 9E9, 9E9, 9E9, 9E9, 9E9]];
	VAR robtarget Openhole_3975 := [[536.36, -24.92, 184.62], [0.183051, 0.683002, 0.683002, -0.183051], [0,0,0,0], [9E9, 9E9, 9E9, 9E9, 9E9, 9E9]];
	VAR robtarget Openhole_3976 := [[536.36, -25.98, 185.23], [0.183051, 0.683002, 0.683002, -0.183051], [0,0,0,0], [9E9, 9E9, 9E9, 9E9, 9E9, 9E9]];
	VAR robtarget Openhole_3977 := [[509.36, -25.98, 185.31], [0.183051, 0.683002, 0.683002, -0.183051], [0,0,0,0], [9E9, 9E9, 9E9, 9E9, 9E9, 9E9]];
	VAR robtarget Openhole_3978 := [[504.36, -25.98, 184.98], [0.191542, 0.68067, 0.691135, -0.149441], [0,0,0,0], [9E9, 9E9, 9E9, 9E9, 9E9, 9E9]];
	VAR robtarget Openhole_3979 := [[492.57, -26.46, 184.39], [0.162281, 0.688233, 0.69773, -0.114771], [0,0,0,0], [9E9, 9E9, 9E9, 9E9, 9E9, 9E9]];
	VAR robtarget Openhole_3980 := [[471.63, -27.19, 183.05], [0.102657, 0.699615, 0.705568, -0.046619], [0,0,0,0], [9E9, 9E9, 9E9, 9E9, 9E9, 9E9]];
	VAR robtarget Openhole_3981 := [[456.18, -27.73, 181.87], [0.053946, 0.705046, 0.70707, 0.007207], [0,0,0,0], [9E9, 9E9, 9E9, 9E9, 9E9, 9E9]];
	VAR robtarget Openhole_3982 := [[455.68, -27.74, 181.83], [0.052306, 0.70517, 0.70705, 0.00894], [0,0,0,0], [9E9, 9E9, 9E9, 9E9, 9E9, 9E9]];
	VAR robtarget Openhole_3983 := [[454.69, -27.73, 181.75], [0.048905, 0.705414, 0.707, 0.012287], [0,0,0,0], [9E9, 9E9, 9E9, 9E9, 9E9, 9E9]];
	VAR robtarget Openhole_3984 := [[454.19, -27.71, 181.71], [0.047157, 0.705533, 0.70697, 0.013913], [0,0,0,0], [9E9, 9E9, 9E9, 9E9, 9E9, 9E9]];
	VAR robtarget Openhole_3985 := [[452.7, -27.62, 181.58], [0.041824, 0.705869, 0.706859, 0.018704], [0,0,0,0], [9E9, 9E9, 9E9, 9E9, 9E9, 9E9]];
	VAR robtarget Openhole_3986 := [[448.72, -27.39, 181.25], [0.027535, 0.70657, 0.706407, 0.031457], [0,0,0,0], [9E9, 9E9, 9E9, 9E9, 9E9, 9E9]];
	VAR robtarget Openhole_3987 := [[448.22, -27.39, 181.21], [0.025833, 0.706635, 0.70633, 0.033143], [0,0,0,0], [9E9, 9E9, 9E9, 9E9, 9E9, 9E9]];
	VAR robtarget Openhole_3988 := [[447.72, -27.4, 181.17], [0.024179, 0.706693, 0.706246, 0.034875], [0,0,0,0], [9E9, 9E9, 9E9, 9E9, 9E9, 9E9]];
	VAR robtarget Openhole_3989 := [[447.22, -27.43, 181.13], [0.022564, 0.706747, 0.706157, 0.036642], [0,0,0,0], [9E9, 9E9, 9E9, 9E9, 9E9, 9E9]];
	VAR robtarget Openhole_3990 := [[445.74, -27.57, 181], [0.017966, 0.706879, 0.705849, 0.042151], [0,0,0,0], [9E9, 9E9, 9E9, 9E9, 9E9, 9E9]];
	VAR robtarget Openhole_3991 := [[442.28, -28.03, 180.69], [0.007743, 0.707064, 0.704938, 0.055337], [0,0,0,0], [9E9, 9E9, 9E9, 9E9, 9E9, 9E9]];
	VAR robtarget Openhole_3992 := [[441.3, -28.17, 180.59], [0.004858, 0.70709, 0.704632, 0.059108], [0,0,0,0], [9E9, 9E9, 9E9, 9E9, 9E9, 9E9]];
	VAR robtarget Openhole_3993 := [[438.84, -28.58, 180.34], [-0.002113, 0.707104, 0.703766, 0.068652], [0,0,0,0], [9E9, 9E9, 9E9, 9E9, 9E9, 9E9]];
	VAR robtarget Openhole_3994 := [[437.87, -28.76, 180.23], [-0.00485, 0.70709, 0.703382, 0.072478], [0,0,0,0], [9E9, 9E9, 9E9, 9E9, 9E9, 9E9]];
	VAR robtarget Openhole_3995 := [[430.08, -30.27, 179.22], [-0.026161, 0.706623, 0.699599, 0.102769], [0,0,0,0], [9E9, 9E9, 9E9, 9E9, 9E9, 9E9]];
	VAR robtarget Openhole_3996 := [[425.17, -30.94, 178.53], [-0.040311, 0.705957, 0.696789, 0.120356], [0,0,0,0], [9E9, 9E9, 9E9, 9E9, 9E9, 9E9]];
	VAR robtarget Openhole_3997 := [[420.22, -31.24, 177.88], [-0.055563, 0.70492, 0.69383, 0.13638], [0,0,0,0], [9E9, 9E9, 9E9, 9E9, 9E9, 9E9]];
	VAR robtarget Openhole_3998 := [[418.24, -31.27, 177.64], [-0.061918, 0.704391, 0.69263, 0.142348], [0,0,0,0], [9E9, 9E9, 9E9, 9E9, 9E9, 9E9]];
	VAR robtarget Openhole_3999 := [[417.74, -31.27, 177.58], [-0.063522, 0.704248, 0.692329, 0.143805], [0,0,0,0], [9E9, 9E9, 9E9, 9E9, 9E9, 9E9]];
	VAR robtarget Openhole_4000 := [[411.78, -31.03, 176.96], [-0.083147, 0.702201, 0.688718, 0.160212], [0,0,0,0], [9E9, 9E9, 9E9, 9E9, 9E9, 9E9]];
	VAR robtarget Openhole_4001 := [[397.86, -29.96, 175.89], [-0.127805, 0.695461, 0.679992, 0.193934], [0,0,0,0], [9E9, 9E9, 9E9, 9E9, 9E9, 9E9]];
	VAR robtarget Openhole_4002 := [[394.33, -29.87, 175.56], [-0.137879, 0.693534, 0.677525, 0.202386], [0,0,0,0], [9E9, 9E9, 9E9, 9E9, 9E9, 9E9]];
	VAR robtarget Openhole_4003 := [[389.33, -29.87, 175.04], [-0.151321, 0.690726, 0.673892, 0.214172], [0,0,0,0], [9E9, 9E9, 9E9, 9E9, 9E9, 9E9]];
	VAR robtarget Openhole_4004 := [[362.33, -29.87, 175.12], [-0.183051, 0.683002, 0.683002, 0.183051], [0,0,0,0], [9E9, 9E9, 9E9, 9E9, 9E9, 9E9]];
	VAR robtarget Openhole_4005 := [[361.41, -38.7, 170.03], [-0.183051, 0.683002, 0.683002, 0.183051], [0,0,0,0], [9E9, 9E9, 9E9, 9E9, 9E9, 9E9]];
	VAR robtarget Openhole_4006 := [[389.31, -38.7, 169.94], [-0.126246, 0.695746, 0.665704, 0.238407], [0,0,0,0], [9E9, 9E9, 9E9, 9E9, 9E9, 9E9]];
	VAR robtarget Openhole_4007 := [[480.22, -38.7, 187.14], [0.165157, 0.687549, 0.706098, -0.03776], [0,0,0,0], [9E9, 9E9, 9E9, 9E9, 9E9, 9E9]];
	VAR robtarget Openhole_4008 := [[488.08, -37.66, 188.24], [0.183899, 0.682775, 0.703985, -0.066368], [0,0,0,0], [9E9, 9E9, 9E9, 9E9, 9E9, 9E9]];
	VAR robtarget Openhole_4009 := [[498.44, -36.73, 189.66], [0.207919, 0.675848, 0.69987, -0.100904], [0,0,0,0], [9E9, 9E9, 9E9, 9E9, 9E9, 9E9]];
	VAR robtarget Openhole_4010 := [[504.37, -36.35, 190.47], [0.221014, 0.671679, 0.696988, -0.119195], [0,0,0,0], [9E9, 9E9, 9E9, 9E9, 9E9, 9E9]];
	VAR robtarget Openhole_4011 := [[504.38, -36.35, 190.47], [0.221026, 0.671675, 0.696985, -0.119212], [0,0,0,0], [9E9, 9E9, 9E9, 9E9, 9E9, 9E9]];
	VAR robtarget Openhole_4012 := [[509.38, -36.35, 191.3], [0.183051, 0.683002, 0.683002, -0.183051], [0,0,0,0], [9E9, 9E9, 9E9, 9E9, 9E9, 9E9]];
	VAR robtarget Openhole_4013 := [[536.38, -36.35, 191.22], [0.183051, 0.683002, 0.683002, -0.183051], [0,0,0,0], [9E9, 9E9, 9E9, 9E9, 9E9, 9E9]];
	VAR robtarget Openhole_4014 := [[536.38, -35.46, 190.71], [0.183051, 0.683002, 0.683002, -0.183051], [0,0,0,0], [9E9, 9E9, 9E9, 9E9, 9E9, 9E9]];
	VAR robtarget Openhole_4015 := [[509.38, -35.46, 190.79], [0.183051, 0.683002, 0.683002, -0.183051], [0,0,0,0], [9E9, 9E9, 9E9, 9E9, 9E9, 9E9]];
	VAR robtarget Openhole_4016 := [[504.37, -35.46, 190], [0.218552, 0.672484, 0.696542, -0.121774], [0,0,0,0], [9E9, 9E9, 9E9, 9E9, 9E9, 9E9]];
	VAR robtarget Openhole_4017 := [[504.37, -35.46, 190], [0.218547, 0.672486, 0.696543, -0.121767], [0,0,0,0], [9E9, 9E9, 9E9, 9E9, 9E9, 9E9]];
	VAR robtarget Openhole_4018 := [[503.88, -35.49, 189.94], [0.217475, 0.672833, 0.696802, -0.120282], [0,0,0,0], [9E9, 9E9, 9E9, 9E9, 9E9, 9E9]];
	VAR robtarget Openhole_4019 := [[492.01, -36.34, 188.4], [0.190421, 0.680984, 0.702255, -0.082694], [0,0,0,0], [9E9, 9E9, 9E9, 9E9, 9E9, 9E9]];
	VAR robtarget Openhole_4020 := [[483.63, -37.25, 187.31], [0.170391, 0.68627, 0.705085, -0.053437], [0,0,0,0], [9E9, 9E9, 9E9, 9E9, 9E9, 9E9]];
	VAR robtarget Openhole_4021 := [[476.28, -38.4, 186.32], [0.152743, 0.690413, 0.706641, -0.025663], [0,0,0,0], [9E9, 9E9, 9E9, 9E9, 9E9, 9E9]];
	VAR robtarget Openhole_4022 := [[475.31, -38.59, 186.19], [0.150422, 0.690922, 0.70677, -0.021823], [0,0,0,0], [9E9, 9E9, 9E9, 9E9, 9E9, 9E9]];
	VAR robtarget Openhole_4023 := [[474.82, -38.7, 186.12], [0.149321, 0.691161, 0.706829, -0.019827], [0,0,0,0], [9E9, 9E9, 9E9, 9E9, 9E9, 9E9]];
	VAR robtarget Openhole_4024 := [[470.42, -38.7, 185.29], [0.135951, 0.693914, 0.707089, -0.004994], [0,0,0,0], [9E9, 9E9, 9E9, 9E9, 9E9, 9E9]];
	VAR robtarget Openhole_4025 := [[470.91, -38.55, 185.35], [0.136975, 0.693713, 0.707071, -0.007113], [0,0,0,0], [9E9, 9E9, 9E9, 9E9, 9E9, 9E9]];
	VAR robtarget Openhole_4026 := [[477.71, -37.2, 186.26], [0.153231, 0.690304, 0.706277, -0.034249], [0,0,0,0], [9E9, 9E9, 9E9, 9E9, 9E9, 9E9]];
	VAR robtarget Openhole_4027 := [[485.08, -36.14, 187.18], [0.171092, 0.686096, 0.704421, -0.061572], [0,0,0,0], [9E9, 9E9, 9E9, 9E9, 9E9, 9E9]];
	VAR robtarget Openhole_4028 := [[493.97, -35.28, 188.28], [0.192432, 0.680419, 0.701109, -0.091906], [0,0,0,0], [9E9, 9E9, 9E9, 9E9, 9E9, 9E9]];
	VAR robtarget Openhole_4029 := [[504.37, -34.58, 189.53], [0.216071, 0.673286, 0.696089, -0.12434], [0,0,0,0], [9E9, 9E9, 9E9, 9E9, 9E9, 9E9]];
	VAR robtarget Openhole_4030 := [[509.37, -34.58, 190.28], [0.183051, 0.683002, 0.683002, -0.183051], [0,0,0,0], [9E9, 9E9, 9E9, 9E9, 9E9, 9E9]];
	VAR robtarget Openhole_4031 := [[536.37, -34.58, 190.2], [0.183051, 0.683002, 0.683002, -0.183051], [0,0,0,0], [9E9, 9E9, 9E9, 9E9, 9E9, 9E9]];
	VAR robtarget Openhole_4032 := [[536.37, -33.69, 189.69], [0.183051, 0.683002, 0.683002, -0.183051], [0,0,0,0], [9E9, 9E9, 9E9, 9E9, 9E9, 9E9]];
	VAR robtarget Openhole_4033 := [[524.37, -33.69, 189.72], [0.183051, 0.683002, 0.683002, -0.183051], [0,0,0,0], [9E9, 9E9, 9E9, 9E9, 9E9, 9E9]];
	VAR robtarget Openhole_4034 := [[509.37, -33.69, 189.77], [0.183051, 0.683002, 0.683002, -0.183051], [0,0,0,0], [9E9, 9E9, 9E9, 9E9, 9E9, 9E9]];
	VAR robtarget Openhole_4035 := [[504.38, -33.69, 189.07], [0.213591, 0.674076, 0.695622, -0.126923], [0,0,0,0], [9E9, 9E9, 9E9, 9E9, 9E9, 9E9]];
	VAR robtarget Openhole_4036 := [[490, -34.71, 187.44], [0.180263, 0.683743, 0.702397, -0.08148], [0,0,0,0], [9E9, 9E9, 9E9, 9E9, 9E9, 9E9]];
	VAR robtarget Openhole_4037 := [[482.1, -35.58, 186.52], [0.160949, 0.688546, 0.705061, -0.053753], [0,0,0,0], [9E9, 9E9, 9E9, 9E9, 9E9, 9E9]];
	VAR robtarget Openhole_4038 := [[475.24, -36.68, 185.7], [0.144232, 0.692241, 0.706565, -0.027687], [0,0,0,0], [9E9, 9E9, 9E9, 9E9, 9E9, 9E9]];
	VAR robtarget Openhole_4039 := [[467.97, -38.24, 184.74], [0.126855, 0.695635, 0.707104, 0.001875], [0,0,0,0], [9E9, 9E9, 9E9, 9E9, 9E9, 9E9]];
	VAR robtarget Openhole_4040 := [[467, -38.47, 184.6], [0.124556, 0.69605, 0.707082, 0.005898], [0,0,0,0], [9E9, 9E9, 9E9, 9E9, 9E9, 9E9]];
	VAR robtarget Openhole_4041 := [[466.52, -38.7, 184.55], [0.123758, 0.696193, 0.707058, 0.008295], [0,0,0,0], [9E9, 9E9, 9E9, 9E9, 9E9, 9E9]];
	VAR robtarget Openhole_4042 := [[462.13, -38.7, 183.72], [0.109748, 0.698538, 0.706723, 0.023285], [0,0,0,0], [9E9, 9E9, 9E9, 9E9, 9E9, 9E9]];
	VAR robtarget Openhole_4043 := [[462.62, -38.48, 183.78], [0.110586, 0.698406, 0.706798, 0.020903], [0,0,0,0], [9E9, 9E9, 9E9, 9E9, 9E9, 9E9]];
	VAR robtarget Openhole_4044 := [[471.3, -36.44, 184.98], [0.131493, 0.694773, 0.706942, -0.015257], [0,0,0,0], [9E9, 9E9, 9E9, 9E9, 9E9, 9E9]];
	VAR robtarget Openhole_4045 := [[478.14, -35.16, 185.77], [0.148128, 0.691418, 0.70585, -0.042135], [0,0,0,0], [9E9, 9E9, 9E9, 9E9, 9E9, 9E9]];
	VAR robtarget Openhole_4046 := [[485.53, -34.21, 186.59], [0.166473, 0.687231, 0.703729, -0.069035], [0,0,0,0], [9E9, 9E9, 9E9, 9E9, 9E9, 9E9]];
	VAR robtarget Openhole_4047 := [[495.44, -33.39, 187.67], [0.190651, 0.68092, 0.699706, -0.102038], [0,0,0,0], [9E9, 9E9, 9E9, 9E9, 9E9, 9E9]];
	VAR robtarget Openhole_4048 := [[504.38, -32.81, 188.6], [0.211099, 0.674861, 0.695147, -0.129503], [0,0,0,0], [9E9, 9E9, 9E9, 9E9, 9E9, 9E9]];
	VAR robtarget Openhole_4049 := [[509.37, -32.81, 189.26], [0.183051, 0.683002, 0.683002, -0.183051], [0,0,0,0], [9E9, 9E9, 9E9, 9E9, 9E9, 9E9]];
	VAR robtarget Openhole_4050 := [[536.37, -32.81, 189.18], [0.183051, 0.683002, 0.683002, -0.183051], [0,0,0,0], [9E9, 9E9, 9E9, 9E9, 9E9, 9E9]];
	VAR robtarget Openhole_4051 := [[536.37, -31.93, 188.67], [0.183051, 0.683002, 0.683002, -0.183051], [0,0,0,0], [9E9, 9E9, 9E9, 9E9, 9E9, 9E9]];
	VAR robtarget Openhole_4052 := [[524.37, -31.93, 188.7], [0.183051, 0.683002, 0.683002, -0.183051], [0,0,0,0], [9E9, 9E9, 9E9, 9E9, 9E9, 9E9]];
	VAR robtarget Openhole_4053 := [[509.37, -31.93, 188.75], [0.183051, 0.683002, 0.683002, -0.183051], [0,0,0,0], [9E9, 9E9, 9E9, 9E9, 9E9, 9E9]];
	VAR robtarget Openhole_4054 := [[504.38, -31.93, 188.13], [0.2086, 0.675637, 0.694661, -0.132084], [0,0,0,0], [9E9, 9E9, 9E9, 9E9, 9E9, 9E9]];
	VAR robtarget Openhole_4055 := [[487.99, -33.03, 186.51], [0.169696, 0.686443, 0.702516, -0.080447], [0,0,0,0], [9E9, 9E9, 9E9, 9E9, 9E9, 9E9]];
	VAR robtarget Openhole_4056 := [[479.58, -33.93, 185.64], [0.148506, 0.691336, 0.705278, -0.050816], [0,0,0,0], [9E9, 9E9, 9E9, 9E9, 9E9, 9E9]];
	VAR robtarget Openhole_4057 := [[473.19, -34.93, 184.95], [0.13252, 0.694578, 0.70661, -0.0265], [0,0,0,0], [9E9, 9E9, 9E9, 9E9, 9E9, 9E9]];
	VAR robtarget Openhole_4058 := [[466.4, -36.39, 184.15], [0.115989, 0.697529, 0.707106, 0.001202], [0,0,0,0], [9E9, 9E9, 9E9, 9E9, 9E9, 9E9]];
	VAR robtarget Openhole_4059 := [[457.75, -38.56, 182.88], [0.094988, 0.700698, 0.706094, 0.037826], [0,0,0,0], [9E9, 9E9, 9E9, 9E9, 9E9, 9E9]];
	VAR robtarget Openhole_4060 := [[457.28, -38.7, 182.8], [0.093864, 0.700849, 0.705979, 0.039924], [0,0,0,0], [9E9, 9E9, 9E9, 9E9, 9E9, 9E9]];
	VAR robtarget Openhole_4061 := [[452.92, -38.7, 181.98], [0.07937, 0.702638, 0.70498, 0.054801], [0,0,0,0], [9E9, 9E9, 9E9, 9E9, 9E9, 9E9]];
	VAR robtarget Openhole_4062 := [[460.54, -36.57, 183.19], [0.097682, 0.700327, 0.706771, 0.021787], [0,0,0,0], [9E9, 9E9, 9E9, 9E9, 9E9, 9E9]];
	VAR robtarget Openhole_4063 := [[467.77, -34.81, 184.1], [0.115243, 0.697653, 0.707054, -0.008643], [0,0,0,0], [9E9, 9E9, 9E9, 9E9, 9E9, 9E9]];
	VAR robtarget Openhole_4064 := [[474.13, -33.64, 184.79], [0.131253, 0.694818, 0.706298, -0.0338], [0,0,0,0], [9E9, 9E9, 9E9, 9E9, 9E9, 9E9]];
	VAR robtarget Openhole_4065 := [[481.53, -32.67, 185.52], [0.15026, 0.690957, 0.704459, -0.061141], [0,0,0,0], [9E9, 9E9, 9E9, 9E9, 9E9, 9E9]];
	VAR robtarget Openhole_4066 := [[491.44, -31.83, 186.49], [0.175487, 0.684985, 0.700722, -0.094805], [0,0,0,0], [9E9, 9E9, 9E9, 9E9, 9E9, 9E9]];
	VAR robtarget Openhole_4067 := [[504.38, -31.04, 187.66], [0.2061, 0.676404, 0.694163, -0.134676], [0,0,0,0], [9E9, 9E9, 9E9, 9E9, 9E9, 9E9]];
	VAR robtarget Openhole_4068 := [[509.37, -31.04, 188.24], [0.183051, 0.683002, 0.683002, -0.183051], [0,0,0,0], [9E9, 9E9, 9E9, 9E9, 9E9, 9E9]];
	VAR robtarget Openhole_4069 := [[536.33, -31.04, 188.16], [0.183051, 0.683002, 0.683002, -0.183051], [0,0,0,0], [9E9, 9E9, 9E9, 9E9, 9E9, 9E9]];
	VAR robtarget Openhole_4070 := [[536.24, -21.49, 182.64], [0.183051, 0.683002, 0.683002, -0.183051], [0,0,0,0], [9E9, 9E9, 9E9, 9E9, 9E9, 9E9]];
	VAR robtarget Openhole_4071 := [[509.35, -21.49, 182.73], [0.183051, 0.683002, 0.683002, -0.183051], [0,0,0,0], [9E9, 9E9, 9E9, 9E9, 9E9, 9E9]];
	VAR robtarget Openhole_4072 := [[504.35, -21.49, 182.61], [0.178553, 0.684192, 0.68817, -0.162551], [0,0,0,0], [9E9, 9E9, 9E9, 9E9, 9E9, 9E9]];
	VAR robtarget Openhole_4073 := [[503.38, -21.52, 182.6], [0.176183, 0.684806, 0.688788, -0.159909], [0,0,0,0], [9E9, 9E9, 9E9, 9E9, 9E9, 9E9]];
	VAR robtarget Openhole_4074 := [[493.89, -21.85, 182.51], [0.151865, 0.690606, 0.694525, -0.132799], [0,0,0,0], [9E9, 9E9, 9E9, 9E9, 9E9, 9E9]];
	VAR robtarget Openhole_4075 := [[487.39, -21.9, 182.35], [0.133567, 0.694377, 0.69792, -0.113609], [0,0,0,0], [9E9, 9E9, 9E9, 9E9, 9E9, 9E9]];
	VAR robtarget Openhole_4076 := [[486.89, -21.89, 182.34], [0.132108, 0.694656, 0.698163, -0.112111], [0,0,0,0], [9E9, 9E9, 9E9, 9E9, 9E9, 9E9]];
	VAR robtarget Openhole_4077 := [[473.4, -21.68, 181.92], [0.0902, 0.70133, 0.703573, -0.070608], [0,0,0,0], [9E9, 9E9, 9E9, 9E9, 9E9, 9E9]];
	VAR robtarget Openhole_4078 := [[465.92, -21.31, 181.67], [0.064753, 0.704136, 0.705526, -0.047252], [0,0,0,0], [9E9, 9E9, 9E9, 9E9, 9E9, 9E9]];
	VAR robtarget Openhole_4079 := [[463.93, -21.12, 181.6], [0.05755, 0.704761, 0.705902, -0.041252], [0,0,0,0], [9E9, 9E9, 9E9, 9E9, 9E9, 9E9]];
	VAR robtarget Openhole_4080 := [[457.02, -21.12, 181.46], [0.034443, 0.706267, 0.706878, -0.017992], [0,0,0,0], [9E9, 9E9, 9E9, 9E9, 9E9, 9E9]];
	VAR robtarget Openhole_4081 := [[456.81, -15.81, 181.07], [0.0157, 0.706932, 0.706226, -0.035275], [0,0,0,0], [9E9, 9E9, 9E9, 9E9, 9E9, 9E9]];
	VAR robtarget Openhole_4082 := [[457.68, -15.38, 181.01], [0.017212, 0.706897, 0.705992, -0.039692], [0,0,0,0], [9E9, 9E9, 9E9, 9E9, 9E9, 9E9]];
	VAR robtarget Openhole_4083 := [[458.51, -14.82, 180.93], [0.018096, 0.706875, 0.705714, -0.044361], [0,0,0,0], [9E9, 9E9, 9E9, 9E9, 9E9, 9E9]];
	VAR robtarget Openhole_4084 := [[460.62, -13.5, 180.7], [0.02081, 0.7068, 0.704896, -0.055867], [0,0,0,0], [9E9, 9E9, 9E9, 9E9, 9E9, 9E9]];
	VAR robtarget Openhole_4085 := [[461.06, -13.27, 180.65], [0.021518, 0.706779, 0.704715, -0.058113], [0,0,0,0], [9E9, 9E9, 9E9, 9E9, 9E9, 9E9]];
	VAR robtarget Openhole_4086 := [[460.89, -17, 181.08], [0.033519, 0.706312, 0.705675, -0.044977], [0,0,0,0], [9E9, 9E9, 9E9, 9E9, 9E9, 9E9]];
	VAR robtarget Openhole_4087 := [[462.52, -15.87, 180.9], [0.035182, 0.706231, 0.705021, -0.054269], [0,0,0,0], [9E9, 9E9, 9E9, 9E9, 9E9, 9E9]];
	VAR robtarget Openhole_4088 := [[462.94, -15.6, 180.85], [0.035684, 0.706206, 0.704841, -0.056565], [0,0,0,0], [9E9, 9E9, 9E9, 9E9, 9E9, 9E9]];
	VAR robtarget Openhole_4089 := [[463.79, -15.08, 180.75], [0.036806, 0.706148, 0.704461, -0.061117], [0,0,0,0], [9E9, 9E9, 9E9, 9E9, 9E9, 9E9]];
	VAR robtarget Openhole_4090 := [[464.66, -14.6, 180.65], [0.038084, 0.70608, 0.704056, -0.065611], [0,0,0,0], [9E9, 9E9, 9E9, 9E9, 9E9, 9E9]];
	VAR robtarget Openhole_4091 := [[465.55, -14.15, 180.54], [0.039547, 0.706, 0.703631, -0.070029], [0,0,0,0], [9E9, 9E9, 9E9, 9E9, 9E9, 9E9]];
	VAR robtarget Openhole_4092 := [[466, -13.94, 180.49], [0.040351, 0.705955, 0.70341, -0.072207], [0,0,0,0], [9E9, 9E9, 9E9, 9E9, 9E9, 9E9]];
	VAR robtarget Openhole_4093 := [[466.46, -13.74, 180.43], [0.041198, 0.705906, 0.703186, -0.074363], [0,0,0,0], [9E9, 9E9, 9E9, 9E9, 9E9, 9E9]];
	VAR robtarget Openhole_4094 := [[467.38, -13.37, 180.32], [0.043033, 0.705796, 0.702724, -0.078603], [0,0,0,0], [9E9, 9E9, 9E9, 9E9, 9E9, 9E9]];
	VAR robtarget Openhole_4095 := [[467.85, -13.2, 180.26], [0.044011, 0.705736, 0.702488, -0.08069], [0,0,0,0], [9E9, 9E9, 9E9, 9E9, 9E9, 9E9]];
	VAR robtarget Openhole_4096 := [[468.32, -13.04, 180.21], [0.045048, 0.70567, 0.702249, -0.082741], [0,0,0,0], [9E9, 9E9, 9E9, 9E9, 9E9, 9E9]];
	VAR robtarget Openhole_4097 := [[469.27, -12.75, 180.1], [0.047226, 0.705528, 0.701762, -0.086777], [0,0,0,0], [9E9, 9E9, 9E9, 9E9, 9E9, 9E9]];
	VAR robtarget Openhole_4098 := [[470.71, -12.36, 179.93], [0.050693, 0.705287, 0.701007, -0.092679], [0,0,0,0], [9E9, 9E9, 9E9, 9E9, 9E9, 9E9]];
	VAR robtarget Openhole_4099 := [[471.19, -12.25, 179.88], [0.051918, 0.705198, 0.700751, -0.094594], [0,0,0,0], [9E9, 9E9, 9E9, 9E9, 9E9, 9E9]];
	VAR robtarget Openhole_4100 := [[471.68, -12.15, 179.82], [0.05318, 0.705104, 0.700494, -0.09648], [0,0,0,0], [9E9, 9E9, 9E9, 9E9, 9E9, 9E9]];
	VAR robtarget Openhole_4101 := [[475.61, -11.57, 179.42], [0.064097, 0.704196, 0.698378, -0.11076], [0,0,0,0], [9E9, 9E9, 9E9, 9E9, 9E9, 9E9]];
	VAR robtarget Openhole_4102 := [[480.09, -11.3, 179.02], [0.077561, 0.70284, 0.695912, -0.125328], [0,0,0,0], [9E9, 9E9, 9E9, 9E9, 9E9, 9E9]];
	VAR robtarget Openhole_4103 := [[482.58, -11.27, 178.82], [0.085315, 0.701941, 0.694508, -0.132885], [0,0,0,0], [9E9, 9E9, 9E9, 9E9, 9E9, 9E9]];
	VAR robtarget Openhole_4104 := [[483.08, -11.27, 178.78], [0.086875, 0.70175, 0.694224, -0.13436], [0,0,0,0], [9E9, 9E9, 9E9, 9E9, 9E9, 9E9]];
	VAR robtarget Openhole_4105 := [[497.54, -11.57, 177.84], [0.130854, 0.694894, 0.685365, -0.173995], [0,0,0,0], [9E9, 9E9, 9E9, 9E9, 9E9, 9E9]];
	VAR robtarget Openhole_4106 := [[498.04, -11.57, 177.8], [0.132254, 0.694629, 0.685029, -0.175315], [0,0,0,0], [9E9, 9E9, 9E9, 9E9, 9E9, 9E9]];
	VAR robtarget Openhole_4107 := [[503.02, -11.41, 177.36], [0.145516, 0.691972, 0.681497, -0.188577], [0,0,0,0], [9E9, 9E9, 9E9, 9E9, 9E9, 9E9]];
	VAR robtarget Openhole_4108 := [[503.51, -11.37, 177.31], [0.146763, 0.691708, 0.681127, -0.189911], [0,0,0,0], [9E9, 9E9, 9E9, 9E9, 9E9, 9E9]];
	VAR robtarget Openhole_4109 := [[504.33, -11.35, 177.24], [0.148896, 0.691252, 0.680535, -0.192022], [0,0,0,0], [9E9, 9E9, 9E9, 9E9, 9E9, 9E9]];
	VAR robtarget Openhole_4110 := [[509.33, -11.35, 176.87], [0.183051, 0.683002, 0.683002, -0.183051], [0,0,0,0], [9E9, 9E9, 9E9, 9E9, 9E9, 9E9]];
	VAR robtarget Openhole_4111 := [[536.33, -11.35, 176.78], [0.183051, 0.683002, 0.683002, -0.183051], [0,0,0,0], [9E9, 9E9, 9E9, 9E9, 9E9, 9E9]];
	VAR robtarget Openhole_4112 := [[536.34, -13.35, 177.94], [0.183051, 0.683002, 0.683002, -0.183051], [0,0,0,0], [9E9, 9E9, 9E9, 9E9, 9E9, 9E9]];
	VAR robtarget Openhole_4113 := [[509.34, -13.35, 178.02], [0.183051, 0.683002, 0.683002, -0.183051], [0,0,0,0], [9E9, 9E9, 9E9, 9E9, 9E9, 9E9]];
	VAR robtarget Openhole_4114 := [[504.34, -13.35, 178.29], [0.154749, 0.689966, 0.682135, -0.186257], [0,0,0,0], [9E9, 9E9, 9E9, 9E9, 9E9, 9E9]];
	VAR robtarget Openhole_4115 := [[498.25, -13.65, 178.77], [0.139113, 0.693288, 0.686451, -0.16966], [0,0,0,0], [9E9, 9E9, 9E9, 9E9, 9E9, 9E9]];
	VAR robtarget Openhole_4116 := [[494.76, -13.69, 178.97], [0.129375, 0.695171, 0.688735, -0.160136], [0,0,0,0], [9E9, 9E9, 9E9, 9E9, 9E9, 9E9]];
	VAR robtarget Openhole_4117 := [[494.26, -13.69, 178.99], [0.127944, 0.695435, 0.689052, -0.158769], [0,0,0,0], [9E9, 9E9, 9E9, 9E9, 9E9, 9E9]];
	VAR robtarget Openhole_4118 := [[482.27, -13.53, 179.56], [0.091582, 0.701151, 0.696006, -0.124805], [0,0,0,0], [9E9, 9E9, 9E9, 9E9, 9E9, 9E9]];
	VAR robtarget Openhole_4119 := [[481.77, -13.53, 179.59], [0.09003, 0.701352, 0.696273, -0.123302], [0,0,0,0], [9E9, 9E9, 9E9, 9E9, 9E9, 9E9]];
	VAR robtarget Openhole_4120 := [[476.28, -13.68, 179.91], [0.073161, 0.703312, 0.699117, -0.105999], [0,0,0,0], [9E9, 9E9, 9E9, 9E9, 9E9, 9E9]];
	VAR robtarget Openhole_4121 := [[474.29, -13.82, 180.05], [0.067223, 0.703904, 0.700101, -0.099291], [0,0,0,0], [9E9, 9E9, 9E9, 9E9, 9E9, 9E9]];
	VAR robtarget Openhole_4122 := [[473.3, -13.93, 180.13], [0.064373, 0.704171, 0.700588, -0.095796], [0,0,0,0], [9E9, 9E9, 9E9, 9E9, 9E9, 9E9]];
	VAR robtarget Openhole_4123 := [[470.86, -19.93, 181.49], [0.076259, 0.702983, 0.703816, -0.068138], [0,0,0,0], [9E9, 9E9, 9E9, 9E9, 9E9, 9E9]];
	VAR robtarget Openhole_4124 := [[487.35, -20.27, 181.75], [0.128331, 0.695364, 0.697086, -0.11862], [0,0,0,0], [9E9, 9E9, 9E9, 9E9, 9E9, 9E9]];
	VAR robtarget Openhole_4125 := [[489.35, -20.27, 181.78], [0.134167, 0.694262, 0.696057, -0.124517], [0,0,0,0], [9E9, 9E9, 9E9, 9E9, 9E9, 9E9]];
	VAR robtarget Openhole_4126 := [[489.85, -20.27, 181.79], [0.135607, 0.693982, 0.695793, -0.125984], [0,0,0,0], [9E9, 9E9, 9E9, 9E9, 9E9, 9E9]];
	VAR robtarget Openhole_4127 := [[499.85, -20.1, 181.82], [0.162753, 0.688122, 0.68998, -0.154687], [0,0,0,0], [9E9, 9E9, 9E9, 9E9, 9E9, 9E9]];
	VAR robtarget Openhole_4128 := [[504.35, -19.88, 181.76], [0.173864, 0.685399, 0.687042, -0.167253], [0,0,0,0], [9E9, 9E9, 9E9, 9E9, 9E9, 9E9]];
	VAR robtarget Openhole_4129 := [[536.35, -19.88, 181.71], [0.183051, 0.683002, 0.683002, -0.183051], [0,0,0,0], [9E9, 9E9, 9E9, 9E9, 9E9, 9E9]];
	VAR robtarget Openhole_4130 := [[536.35, -19.19, 181.31], [0.183051, 0.683002, 0.683002, -0.183051], [0,0,0,0], [9E9, 9E9, 9E9, 9E9, 9E9, 9E9]];
	VAR robtarget Openhole_4131 := [[509.35, -19.19, 181.39], [0.183051, 0.683002, 0.683002, -0.183051], [0,0,0,0], [9E9, 9E9, 9E9, 9E9, 9E9, 9E9]];
	VAR robtarget Openhole_4132 := [[504.35, -19.19, 181.39], [0.17183, 0.685911, 0.686543, -0.169287], [0,0,0,0], [9E9, 9E9, 9E9, 9E9, 9E9, 9E9]];
	VAR robtarget Openhole_4133 := [[495.63, -19.51, 181.52], [0.14956, 0.691109, 0.692108, -0.144867], [0,0,0,0], [9E9, 9E9, 9E9, 9E9, 9E9, 9E9]];
	VAR robtarget Openhole_4134 := [[490.13, -19.56, 181.51], [0.134196, 0.694256, 0.695235, -0.12903], [0,0,0,0], [9E9, 9E9, 9E9, 9E9, 9E9, 9E9]];
	VAR robtarget Openhole_4135 := [[489.63, -19.56, 181.51], [0.132751, 0.694534, 0.695503, -0.127573], [0,0,0,0], [9E9, 9E9, 9E9, 9E9, 9E9, 9E9]];
	VAR robtarget Openhole_4136 := [[470.13, -19.24, 181.34], [0.071633, 0.703469, 0.703822, -0.068074], [0,0,0,0], [9E9, 9E9, 9E9, 9E9, 9E9, 9E9]];
	VAR robtarget Openhole_4137 := [[469.63, -19.24, 181.34], [0.070009, 0.703633, 0.703979, -0.06644], [0,0,0,0], [9E9, 9E9, 9E9, 9E9, 9E9, 9E9]];
	VAR robtarget Openhole_4138 := [[469.13, -19.24, 181.34], [0.068372, 0.703793, 0.70413, -0.064811], [0,0,0,0], [9E9, 9E9, 9E9, 9E9, 9E9, 9E9]];
	VAR robtarget Openhole_4139 := [[466.63, -19.31, 181.35], [0.060419, 0.704521, 0.704858, -0.05635], [0,0,0,0], [9E9, 9E9, 9E9, 9E9, 9E9, 9E9]];
	VAR robtarget Openhole_4140 := [[466.13, -19.31, 181.35], [0.058784, 0.704659, 0.704989, -0.054683], [0,0,0,0], [9E9, 9E9, 9E9, 9E9, 9E9, 9E9]];
	VAR robtarget Openhole_4141 := [[465.64, -19.33, 181.35], [0.057185, 0.704791, 0.70512, -0.052976], [0,0,0,0], [9E9, 9E9, 9E9, 9E9, 9E9, 9E9]];
	VAR robtarget Openhole_4142 := [[464.64, -19.38, 181.35], [0.054064, 0.705037, 0.705374, -0.049474], [0,0,0,0], [9E9, 9E9, 9E9, 9E9, 9E9, 9E9]];
	VAR robtarget Openhole_4143 := [[464.14, -19.42, 181.36], [0.052543, 0.705152, 0.705497, -0.047682], [0,0,0,0], [9E9, 9E9, 9E9, 9E9, 9E9, 9E9]];
